(* CoDeSys 2.3.9.16 project: PLC_OPEN_test.pro *)
(* Libraries: SysLibTargetVisu.lib 22.7.09 19:44:32, ANALYZATION.LIB 22.7.09 19:44:32, SysLibSockets.lib 22.7.09 19:44:32, SysLibCom.lib 22.7.09 19:44:32, SysLibTime.lib 22.7.09 19:44:32, AD_Convertor.lib 8.4.16 09:37:26, CPAC_TCP.lib 26.6.14 15:50:29, Standard.lib 22.7.09 19:44:32, IecSfc.lib 22.7.09 19:44:32, CPAC GUC-X00-TPX.lib 28.10.10 10:45:18, SysLibMem.lib 22.7.09 19:44:32, SysTaskInfo.lib 22.7.09 19:44:32, SYSLIBCALLBACK.LIB 22.7.09 19:44:32, 3S_CANopenMaster.lib 28.10.13 11:32:40, 3S_CANopenManager.lib 28.10.13 11:32:40, 3S_CanDrv.lib 28.10.13 11:32:40 *)

(* Task configuration *)
TASK PLC_PRG_TASK (PRIORITY := 1, INTERVAL := T#30ms);
	PLC_PRG
	RT_Manager
	TiltManager
	LiftManager
END_TASK
TASK VISU_TASK (PRIORITY := 15, INTERVAL := T#800ms);
	MAINTARGETVISU_PAINT_CODE
END_TASK
TASK SensorRead (PRIORITY := 10, INTERVAL := T#30ms);
	SensorRead();
END_TASK
TASK VISU_INPUT_TASK (PRIORITY := 14, INTERVAL := T#50ms);
	MAINTARGETVISU_INPUT_CODE
END_TASK

(* Global variable list: CanOpen implicit Variables *)
VAR_GLOBAL CONSTANT
	MAX_CTRLINDEX : INT := 0;
END_VAR
VAR_GLOBAL CONSTANT
	USE_CANOPEN_NODES : BOOL := TRUE;
	MAX_MASTERINDEX : INT := 0;
	MAX_NODEINDEX : INT := 1;
	MAX_SDOINDEX : INT := 65;
	MAX_PDOINDEX_RX : INT := 7;
	MAX_PDOINDEX_TX : INT := 7;
	MAX_MASTER_ODENTRY_IDX : INT := 0;
END_VAR
VAR_GLOBAL
	pCANopenMaster : ARRAY[0..MAX_MASTERINDEX] OF CanOpenMaster;
	pCanOpenNode : ARRAY[0..MAX_NODEINDEX] OF CanOpenNode;
	pCanOpenSDO : ARRAY[0..MAX_SDOINDEX] OF CanOpenSDO;
	pCanOpenPDO_Rx : ARRAY[0..MAX_PDOINDEX_RX] OF CanOpenPDO_Rx;
	pCanOpenPDO_Tx : ARRAY[0..MAX_PDOINDEX_TX] OF CanOpenPDO_Tx;
	 ODMEntries: ARRAY[0..MAX_MASTER_ODENTRY_IDX] OF CanOpenODEntry;
END_VAR

(* Global variable list: CANopen_MC_GLB *)
VAR_GLOBAL
	g_CAN_udiStationAmount:UDINT;	(*driver amount on the bus*)
	g_CAN_arAxis: ARRAY [1..255] OF TAxisStatus;	(*0:no mode 1:PP mode 2:PV mode 3:TC mode 4:Homing*)
END_VAR

(* Global variable list: Global_Variables *)
VAR_GLOBAL
	ComHandle: DWORD;
	byRead:ARRAY[1..16]OF BYTE;
	diSocket: DINT:= SOCKET_INVALID;(*SOCKET_INVALID=-1,DINT类型,FFFFFFFF,*)
	xRelativeExe1,xRelativeExe2: BOOL;
	xPowerOn1,xPowerOn2: BOOL;
	xPowerOff1,xPowerOff2: BOOL;
	xStop1,xStop2: BOOL;
	xVelocityExe1,xVelocityExe2: BOOL;
	xReset1,xReset2: BOOL;
	diVelocity1: UDINT:=20000;
	diPosition1,diPosition2: DINT;
	diVelocity2: UDINT:= 20000;
	diVelocity_jog1,diVelocity_jog2: DINT;
	Acc,Dec:DINT;(*加/减速度*)
	ENC_POS1: LREAL;(*病床磁条编码器读数*)
	ENC_POS2: LREAL;(*旋转部编码器读数*)
	ENC_Value: DINT;(*检测到INDEX信号时外部编码器的读数*)
	Client0,Client1,Client2: CLIENT_ACCEPT;
	LiftSpeed:UINT;
	Input_Value:DINT;
	Move_Height:REAL;
	Move_Angle:REAL;

	gLastLiftAngle:REAL;
	gLiftMotionState:UINT:=0;
END_VAR

(* Data type *)
TYPE TAxisStatus :
STRUCT
	usiAxis:USINT;			(*Axis address*)
	usiCurrentMode:USINT;	(*current motion mode*)


END_STRUCT
END_TYPE

(* POU 主程序/PLC_PRG, ST *)
PROGRAM PLC_PRG
VAR
	uiPort: UINT:= 5000;
	bActive: BOOL:=TRUE;
	ON:BOOL:=TRUE;
	RO:ARRAY [1..5] OF BYTE:=16#52,16#4F,16#00,16#5C,16#2D;
	RC:ARRAY [1..7] OF BYTE:=16#52,16#43,16#01,16#00,16#FF,16#31,16#8D;
	ROON,RCON:UINT;
	ComUseTimer:TON;
	cs:COMSETTINGS;(*RS232通讯*)
	bInit,bExit,open,close: BOOL;
	ComFilter:ComFilter;

	byReadRO:ARRAY [1..16] OF BYTE;
	ENC_Status:INT;
	LastIndexVelue:DINT;
	Offset: ARRAY [1..10] OF DINT;
	i:DINT;
	asda: DINT;
END_VAR
IF ON THEN(*寄存器初始化*)
	RegisterCallbacks();
	bInit:=TRUE;
	ON:=FALSE;
END_IF
IF bInit  THEN(* Open COM interface *)
	bInit:=FALSE;bExit:=FALSE;
	cs.	Port:=COM2;
	cs.dwBaudRate:=38400;
	cs.byParity:=0;
	cs.byStopBits:=1;
	cs.dwBufferSize:=1024;
	ComHandle := SysComOpen(cs.Port);
	IF ComHandle<> INVALID_HANDLE THEN(* INVALID_HANDLED，常数，代表32位FFFFFFFF*)
		open := SysComSetSettings(ComHandle, ADR(cs));(*OPEN=1，串口处于正常打开状态*)
		IF open THEN
			close:=FALSE;
		END_IF
	ELSE
		bExit:=TRUE;
	END_IF
END_IF
IF bExit THEN(* Close COM interface *)
	bExit:=FALSE;bInit:=FALSE;
	close := SysComClose(ComHandle);(*close=1，串口处于关闭状态*)
	ComHandle:=0;
	IF close THEN
		open:=FALSE;
	END_IF
END_IF
ComFilter();
CASE ROON OF(*ROON：RO指令发送和接收具体步骤*)
0:	ComUseTimer(IN:=TRUE,PT:=t#3s);
	IF ComUseTimer.Q THEN
		ROON:=1;
		ComUseTimer(IN:=FALSE,PT:=t#3s);
	END_IF
1:	SysComWrite(ComHandle, ADR(RO), 5, 5);	(*发送RO指令*)
	ROON:=2;
2:	IF byRead[1]=16#52 AND byRead[2]=16#4F THEN
		byReadRO:=byRead;
		ROON:=3;
		ComUseTimer(IN:=FALSE,PT:=t#3s);
	END_IF
	ComUseTimer(IN:=TRUE,PT:=t#3s);
	IF ComUseTimer.Q THEN
		ROON:=99;
		ComUseTimer(IN:=FALSE,PT:=t#3s);
	END_IF
3:	IF   byReadRO[1]=16#52 AND byReadRO[2]=16#4F AND byReadRO[3]=16#06 THEN(*判断接收每个字节的内容，该语句判断为正确的回码*)
		ROON:=4;
		RCON:=1;			(*ROON为4证明RO指令发送成功,RCON=1，开始发送RC指令*)
	ELSIF byReadRO[1]=16#52 AND byReadRO[2]=16#4F AND byReadRO[3]<>16#06THEN(*判断接收前三个字节的内容，该语句判断为错误的回码*)
		ROON:=100;(*步骤停止在100并报错*)
	END_IF
END_CASE
CASE RCON OF
1:	SysComWrite(ComHandle, ADR(RC), 7, 5);(*发送RC指令*)
	RCON:=2;
2:	ComUseTimer(IN:=TRUE,PT:=t#250ms);(*定时器*)
	IF ComUseTimer.Q THEN(*定时250ms到，发送一次RC指令*)
		RCON:=1;
		ComUseTimer(IN:=FALSE,PT:=t#250ms);(*定时器*)
	END_IF
END_CASE
IF bActive THEN
	IF diSocket = SOCKET_INVALID THEN
		diSocket := TcpServerOpenSocket(uiPort, 3);(*TCP/IP设置，按F1可查看功能解释*)
	ELSE
		IF Client0.diSocket = SOCKET_INVALID THEN
			Client0:= TcpServerWaitForConnect(diSocket, 200);
		END_IF
		IF Client1.diSocket = SOCKET_INVALID THEN
			Client1:= TcpServerWaitForConnect(diSocket, 200);
		END_IF
		IF Client2.diSocket = SOCKET_INVALID THEN
			Client2:= TcpServerWaitForConnect(diSocket, 200);
		END_IF
	END_IF
ELSE
	IF diSocket <> SOCKET_INVALID THEN(*关闭服务器连接端口*)
		CloseSocket(ADR(diSocket));
		IF Client0.diSocket <> SOCKET_INVALID THEN
			CloseSocket(ADR(Client0.diSocket));
			Client0.stIPAddress:= '';
		END_IF
		IF Client1.diSocket <> SOCKET_INVALID THEN
			CloseSocket(ADR(Client1.diSocket));
			Client1.stIPAddress:= '';
		END_IF
		IF Client2.diSocket <> SOCKET_INVALID THEN
			CloseSocket(ADR(Client2.diSocket));
			Client2.stIPAddress:= '';
		END_IF
	END_IF
END_IF
GT_GetEncPos(9, ADR(ENC_POS1), 1, 0);	(*读取编码器位置：病床平移编码器*)
GT_GetEncPos(4, ADR(ENC_POS2), 1, 0);	(*读取编码器位置：机架旋转部编码器*)
GT_SetCaptureMode(4,CAPTURE_INDEX);	(*F1查询函数定义*)
GT_GetCaptureStatus(4, ADR(ENC_Status), ADR(ENC_Value), 1,0);(*读取编码器捕获状态：读取机架编码器Index信号*)
GT_GetDi(MC_GPI,ADR(Input_Value));(*读取端子板数字输入口信息*)
IF ENC_Value>0AND(ENC_Value/5760)<1 AND i<=10THEN
	LastIndexVelue:=ENC_Value;
ELSIF (ENC_Value/5760)>1 AND i<=10THEN
	IF ENC_Value<>LastIndexVelue  THEN
		IF ((ENC_Value-LastIndexVelue)<>5760)THEN
			i:=i+1;
			Offset[i]:=ENC_Value-LastIndexVelue;
			LastIndexVelue:=ENC_Value;
		ELSE
			LastIndexVelue:=ENC_Value;
		END_IF
	END_IF
END_IF
END_PROGRAM

(* POU PLCOpen_CAN2.3/串口通讯/ComFilter, ST *)
FUNCTION_BLOCK ComFilter
VAR_INPUT
END_VAR
VAR_OUTPUT
END_VAR
VAR
	NullArray,Buffer,MyBuffer:ARRAY [1..16] OF BYTE;
	ComRecieveBytes,MyRecieveBytes:DWORD;
	i:UINT:=0;
	j,k,l,m,n:UINT;
END_VAR
IF ComHandle<> INVALID_HANDLE THEN
	ComRecieveBytes:=SysComRead(ComHandle,ADR(Buffer) , 12, 1);(*串口接收*)
	IF i=1 THEN
		IF  ComRecieveBytes=4 THEN
			IF	Buffer[1]<>16#47 THEN
				MyBuffer[2]:=Buffer[1];
				MyBuffer[3]:=Buffer[2];
				MyBuffer[4]:=Buffer[3];
				MyBuffer[5]:=Buffer[4];
				byRead:=MyBuffer;
				MyBuffer:=NullArray;
				i:=0;

			(*ELSE
				MyBuffer:=NullArray;
				i:=0;*)
			END_IF
		ELSIF ComRecieveBytes>4  THEN
			IF	Buffer[1]=16#47 THEN
				MyBuffer[2]:=Buffer[1];
				MyBuffer[3]:=Buffer[2];
				MyBuffer[4]:=Buffer[3];
				MyBuffer[5]:=Buffer[4];
				MyBuffer[6]:=Buffer[5];
				MyBuffer[7]:=Buffer[6];
				MyBuffer[8]:=Buffer[7];
				MyBuffer[9]:=Buffer[8];
				byRead:=MyBuffer;
				MyBuffer:=NullArray;
				i:=0;
			(*ELSE
				MyBuffer:=NullArray;
				i:=0;*)
			END_IF
		END_IF
	ELSIF i=2 THEN
		IF  ComRecieveBytes=5-MyRecieveBytes THEN
			MyBuffer[MyRecieveBytes+1]:=Buffer[1];
			MyBuffer[MyRecieveBytes+2]:=Buffer[2];
			MyBuffer[MyRecieveBytes+3]:=Buffer[3];
			MyBuffer[MyRecieveBytes+4]:=Buffer[4];
			MyBuffer[MyRecieveBytes+5]:=Buffer[5];
			byRead:=MyBuffer;
			MyBuffer:=NullArray;
			MyRecieveBytes:=0;
			i:=0;
		(*ELSE
			MyBuffer:=NullArray;
			MyRecieveBytes:=0;
			i:=0;*)
		END_IF
	ELSIF i=3 THEN
		IF  ComRecieveBytes=9-MyRecieveBytes THEN
			MyBuffer[MyRecieveBytes+1]:=Buffer[1];
			MyBuffer[MyRecieveBytes+2]:=Buffer[2];
			MyBuffer[MyRecieveBytes+3]:=Buffer[3];
			MyBuffer[MyRecieveBytes+4]:=Buffer[4];
			MyBuffer[MyRecieveBytes+5]:=Buffer[5];
			MyBuffer[MyRecieveBytes+6]:=Buffer[6];
			MyBuffer[MyRecieveBytes+7]:=Buffer[7];
			byRead:=MyBuffer;
			MyBuffer:=NullArray;
			MyRecieveBytes:=0;
			i:=0;
		(*ELSE
			MyBuffer:=NullArray;
			MyRecieveBytes:=0;
			i:=0;*)
		END_IF
	END_IF
	IF i=0 AND ComRecieveBytes=1 AND Buffer[1]=16#52 THEN
		MyBuffer:=Buffer;
		Buffer:=NullArray;
		i:=1;
	ELSIF i=0 AND ComRecieveBytes>1AND ComRecieveBytes<5 AND Buffer[1]=16#52THEN
		IF  Buffer[2]<>16#47 THEN
			MyBuffer:=Buffer;
			MyRecieveBytes:=ComRecieveBytes;
			Buffer:=NullArray;
			i:=2;
		ELSIF	 Buffer[2]=16#47 THEN
			MyBuffer:=Buffer;
			MyRecieveBytes:=ComRecieveBytes;
			Buffer:=NullArray;
			i:=3;
		END_IF
	ELSIF	i=0 AND ComRecieveBytes=5 AND Buffer[1]=16#52 THEN
		IF Buffer[2]<>16#47 THEN
			byRead:=Buffer;
			Buffer:=NullArray;
		ELSIF  Buffer[2]=16#47 THEN
			MyBuffer:=Buffer;
			MyRecieveBytes:=ComRecieveBytes;
			Buffer:=NullArray;
			i:=3;
		END_IF
	ELSIF  i=0 AND ComRecieveBytes>5 AND ComRecieveBytes<9  AND Buffer[1]=16#52 AND  Buffer[2]=16#47THEN
		MyBuffer:=Buffer;
		MyRecieveBytes:=ComRecieveBytes;
		Buffer:=NullArray;
		i:=3;
	ELSIF i=0 AND ComRecieveBytes=9  AND Buffer[1]=16#52 AND  Buffer[2]=16#47THEN
			byRead:=Buffer;
			Buffer:=NullArray;
	END_IF
END_IF
END_FUNCTION_BLOCK

(* POU 子程序/RT_Manager, ST *)
PROGRAM RT_Manager
VAR
	fbRelMove1,fbRelMove2: MC_MoveRelative;
	fbPower1,fbPower2: MC_Power;
	fbStop1,fbStop2: MC_Stop;
	fbVelMove1,fbVelMove2:MC_MoveVelocity;
	fbReset1,fbReset2: MC_Reset;
	LanNullArray,abyRecvRaw,abyRecv,HeartBeat: ARRAY [1..256] OF BYTE;
	diReceived:DINT;
	diRotateHomestep,diRotateJogstep,diRotateMovetostep,diRotateStopstep:UINT;
	diTraverseHomestep,diTraverseJogstep,diTraverseMovetostep,diTraverseStopstep:UINT;
	SizeOfMsg:INT;
	RotateFirstPos,FirstIndexPos:DINT;
	TraverseFirstPos:DINT;
	TargetPosition:LREAL;
	str1: STRING(50):= 'HOME ROTATE;ACK@';str2: STRING(50):= 'HOME ROTATE;UNDERWAY@';str3: STRING(50):= 'HOME ROTATE;COMPLETED@';str4: STRING(50):= 'HOME ROTATE; FAILED=';
	str5: STRING(50):= 'JOG ROTATE;ACK@';str6: STRING(50):= 'JOG ROTATE;UNDERWAY@';str7: STRING(50):= 'JOG ROTATE;COMPLETED@';str8: STRING(50):= 'JOG ROTATE;FAILED=';
	str9: STRING(50):= 'MOVETO ROTATE;ACK@';str10: STRING(50):= 'MOVETO ROTATE;UNDERWAY@';str11: STRING(50):= 'MOVETO ROTATE;COMPLETED@';str12: STRING(50):= 'MOVETO ROTATE;FAILED=';
	str13: STRING(50):= 'STOP ROTATE;ACK@';str14: STRING(50):= 'STOP ROTATE;UNDERWAY@';str15: STRING(50):= 'STOP ROTATE;COMPLETED@';str16: STRING(50):= 'JOG ROTATE;STOPPED@';str17: STRING(50):= 'STOP ROTATE;FAILED=';
	str25: STRING(50):= 'RESET ROTATE;COMPLETED@';str26: STRING(50):= 'RESET ROTATE;FAILED=';
	str30: STRING(50):='HOME ROTATE;STOPPED@';str31: STRING(50):= 'MOVETO ROTATE;STOPPED@';str32: STRING(50):= 'GET ROTATE;COMPLETED;COUNTER =';

	str51: STRING(50):= 'HOME TRAVERSE;ACK@';str52: STRING(50):= 'HOME TRAVERSE;UNDERWAY@';str53: STRING(50):= 'HOME TRAVERSE;COMPLETED@';str54: STRING(50):= 'HOME TRAVERSE; FAILED=';
	str55: STRING(50):= 'JOG TRAVERSE;ACK@';str56: STRING(50):= 'JOG TRAVERSE;UNDERWAY@';str57: STRING(50):= 'JOG TRAVERSE;COMPLETED@';str58: STRING(50):= 'JOG TRAVERSE;FAILED=1@';
	str59: STRING(50):= 'MOVETO TRAVERSE;ACK@';str60: STRING(50):= 'MOVETO TRAVERSE;UNDERWAY@';str61: STRING(50):= 'MOVETO TRAVERSE;COMPLETED@';str62: STRING(50):= 'MOVETO TRAVERSE;FAILED=1@';
	str63: STRING(50):= 'STOP TRAVERSE;ACK@';str64: STRING(50):= 'STOP TRAVERSE;UNDERWAY@';str65: STRING(50):= 'STOP TRAVERSE;COMPLETED@';str66: STRING(50):= 'JOG TRAVERSE;STOPPED@';
	str67: STRING(50):= 'MOVETO TRAVERSE;STOPPED@';str68: STRING(50):= 'HOME TRAVERSE;STOPPED@'; str69: STRING(50):= 'STOP TRAVERSE;FAILED=';
	str73: STRING(50):= 'SET TRAVERSE;COMPLETED@';str74: STRING(50):= 'SET TRAVERSE;FAILED=';

	str77: STRING(50):= 'RESET TRAVERSE;COMPLETED@';str78: STRING(50):= 'RESET TRAVERSE;FAILED=';str79:STRING(50):='JOG TRAVERSE;FAILED=Forward sw Limit@';
	str80:STRING(50):='JOG TRAVERSE;FAILED=Reverse sw Limit@';
	i,j,k,SecondColonPos: INT;
	Temp,Temp1,Temp2,Temp3: STRING;
	RotatePosition,RotateSpeed,RotateTurns,TraversePosition,TraverseSpeed: STRING;
	Horz_Limit_Home,Horz_Limit_In,Horz_Limit_Out:UINT;
	RotateUseTimer1,RotateUseTimer2,RotateUseTimer3,TraverseUseTimer1,TraverseUseTimer2,TraverseUseTimer3:TON;(*信息处理超时*)
	MoveOverTime,AutoSendMsgDelay,HeartBeatTimer:TON;
	AutoSendMsgStep:UINT:=0;
	HeartBeatStep,HeartBeatCounts: INT;
	EmergencyStop: INT;
	OneAngleToPulse: LREAL:=323.9;
END_VAR
IF	 Client0.diSocket <> SOCKET_INVALID THEN
	diReceived:= TcpReceiveData(Client0.diSocket, ADR(abyRecvRaw), SIZEOF(abyRecvRaw), 10);
	IF diReceived>0 THEN
		IF abyRecvRaw[1]=16#52 AND abyRecvRaw[2]=16#54 AND diReceived=22THEN
			HeartBeat:=abyRecvRaw;
			abyRecvRaw:=LanNullArray;
		ELSIF (abyRecvRaw[1]<>16#52 OR abyRecvRaw[2]<>16#54) AND( abyRecvRaw[diReceived-5]<>16#42 OR abyRecvRaw[diReceived-4]<>16#45 OR abyRecvRaw[diReceived-3]<>16#41 OR abyRecvRaw[diReceived-2]<>16#54)THEN
			SizeOfMsg:=DINT_TO_INT(diReceived-2);
			abyRecv:=abyRecvRaw;
			abyRecvRaw:=LanNullArray;
		ELSIF abyRecvRaw[1]=16#52 AND abyRecvRaw[2]=16#54 AND diReceived<>22THEN
			FOR i:=1TO (DINT_TO_INT(diReceived)) BY 1 DO
				IF i<=20 THEN
					HeartBeat[i]:=abyRecvRaw[i];
				END_IF
				IF i>=23 THEN
					abyRecv[i-22]:=abyRecvRaw[i];
				END_IF
				IF  i=diReceived THEN
					abyRecvRaw:=LanNullArray;
				END_IF
			END_FOR
			SizeOfMsg:=DINT_TO_INT(diReceived-24);
		ELSIF abyRecvRaw[1]<>16#52 AND abyRecvRaw[2]<>16#54 AND abyRecvRaw[diReceived-5]=16#42 AND abyRecvRaw[diReceived-4]=16#45 AND abyRecvRaw[diReceived-3]=16#41 AND abyRecvRaw[diReceived-2]=16#54THEN
			FOR i:=1 TO (DINT_TO_INT(diReceived-24))  BY 1 DO
				abyRecv[i]:=abyRecvRaw[i];
			END_FOR
			FOR i:=1 TO 20 BY 1 DO
				HeartBeat[i]:=abyRecvRaw[diReceived-22+i];
			END_FOR
			SizeOfMsg:=DINT_TO_INT(diReceived-24);
			abyRecvRaw:=LanNullArray;
		END_IF
		(*Heart Beat*)
		IF HeartBeat[1]=16#52 AND HeartBeat[2]=16#54 AND HeartBeat[3]=16#4D AND HeartBeat[4]=16#61 AND HeartBeat[5]=16#6E AND HeartBeat[6]=16#61 AND  HeartBeat[7]=16#67 AND HeartBeat[8]=16#65 AND HeartBeat[9]=16#72 THEN
			HeartBeatStep:=1;
			HeartBeatCounts:=HeartBeatCounts+1;
		END_IF
	(*Rotate:版本信息*)
		IF abyRecv[1]=86 AND abyRecv[2]=69AND abyRecv[3]=82 AND abyRecv[4]=83AND abyRecv[5]=73AND abyRecv[6]=79AND abyRecv[7]=78AND abyRecv[8]=32AND abyRecv[9]=82AND abyRecv[10]=79AND abyRecv[11]=84AND abyRecv[12]=65AND abyRecv[13]=84AND abyRecv[14]=69THEN
			Temp:='';
			Temp:='VERSION ROTATE;<version STRING>@';
			TcpSendData(Client0.diSocket, ADR(Temp), LEN(Temp), 10);
			abyRecv:=LanNullArray;
		END_IF
	(*Traverse：获取版本信息*)
		IF((abyRecv[1]=86)AND(abyRecv[2]=69)AND(abyRecv[3]=82)AND(abyRecv[4]=83)AND(abyRecv[5]=73)AND(abyRecv[6]=79)AND(abyRecv[7]=78)AND(abyRecv[8]=32)AND(abyRecv[9]=84 ) AND(abyRecv[10]=82) AND(abyRecv[11]=65 ) AND(abyRecv[12]=86) AND(abyRecv[13]=69) AND(abyRecv[14]=82) AND(abyRecv[15]=83) AND(abyRecv[16]=69) )THEN
			Temp:='';
			Temp:='VERSION TRAVERSE;<version STRING>@';
			TcpSendData(Client0.diSocket, ADR(Temp), LEN(Temp), 0);
			abyRecv:=LanNullArray;
		END_IF
		IF diRotateStopstep=0 THEN
		(*Rotate:Stop动作*)
			IF abyRecv[1]=83AND abyRecv[2]=84AND abyRecv[3]=79 AND abyRecv[4]=80 AND abyRecv[5]=32AND abyRecv[6]=82 AND abyRecv[7]=79AND abyRecv[8]=84AND abyRecv[9]=65AND abyRecv[10]=84AND abyRecv[11]=69 THEN(*判断为Gantry stop命令*)
				TcpSendData(Client0.diSocket, ADR(str13), LEN(str13), 10);(*通过客户端0发送字符串13（STOP ROTATE;ACK）*)
				IF  diRotateJogstep>0 THEN(*如果JOG动作正在执行*)
					diRotateStopstep:=1;diRotateJogstep:=0;xVelocityExe1:=FALSE;
					TcpSendData(Client0.diSocket, ADR(str16), LEN(str16), 10);
				ELSIF  diRotateHomestep>0 THEN(*如果HOME动作正在执行*)
					diRotateStopstep:=20;diRotateHomestep:=0;
					TcpSendData(Client0.diSocket, ADR(str30), LEN(str30), 10);
				ELSIF diRotateMovetostep>0 THEN(*如果MOVETO动作正在执行*)
					diRotateStopstep:=30;diRotateMovetostep:=0;
					TcpSendData(Client0.diSocket, ADR(str31), LEN(str31), 10);
				ELSIF diRotateHomestep=0 AND diRotateMovetostep=0 AND diRotateJogstep=0 THEN(*如果没有任何动作正在执行*)
					diRotateStopstep:=40;
				END_IF
				abyRecv:=LanNullArray;
			ELSIF diRotateHomestep=0 AND diRotateMovetostep=0 AND (diRotateJogstep=0OR diRotateJogstep=4)THEN
			(*Rotate:Home动作*)
				IF abyRecv[1]=72 AND abyRecv[2]=79AND abyRecv[3]=77 AND abyRecv[4]=69 AND abyRecv[5]=32AND abyRecv[6]=82 AND abyRecv[7]=79AND abyRecv[8]=84AND abyRecv[9]=65AND abyRecv[10]=84AND abyRecv[11]=69THEN
					IF ENC_Value<ENC_POS2 OR (ENC_Value=0 AND ENC_POS2 =0)THEN(*满足任一条件：上电后机架已转动过，当前不在Index位置或者系统刚上电机架未转动过*)
						FirstIndexPos:=ENC_Value;(*记录当前滑环编码器index读数*)
						diVelocity_jog1:=-4000;Acc:=4000;Dec:=1000;
						xVelocityExe1:=TRUE;diRotateHomestep:=1;
					ELSIF ENC_Value=ENC_POS2 AND ENC_Value<>0 AND ENC_POS2 <>0THEN(*满足2个条件：1、当前处在在Index位置2、系统上电后机架已转动过 *)
						diRotateHomestep:=3;(*机架不需要旋转，直接回COMPLETE*)
					END_IF
					TcpSendData(Client0.diSocket, ADR(str1), LEN(str1), 10);
					TcpSendData(Client0.diSocket, ADR(str2), LEN(str2), 10);
					abyRecv:=LanNullArray;
			(*Rotate:Moveto动作*)
				ELSIF  abyRecv[1]=77 AND abyRecv[2]=79AND abyRecv[3]=86 AND abyRecv[4]=69AND abyRecv[5]=84AND abyRecv[6]=79AND abyRecv[7]=32AND abyRecv[8]=82AND abyRecv[9]=79AND abyRecv[10]=84AND abyRecv[11]=65AND abyRecv[12]=84 AND abyRecv[13]=69THEN
					Temp1:='';
					FOR j:=1 TO SizeOfMsg DO
						Temp1:=CONCAT(Temp1,ASCII_TO_STRING(abyRecv[j]));(*将命令内容转换为字符串存放在Temp1中*)
					END_FOR;
					TargetPosition:=STRING_TO_LREAL (DELETE(Temp1,24,1));(*目标位置*)
					IF	GR_POS(ENC_Value,ENC_POS2)>0 AND GR_POS(ENC_Value,ENC_POS2)<888.8 THEN
						IF (TargetPosition-GR_POS(ENC_Value,ENC_POS2))>5.0 AND (TargetPosition<>0) THEN(*如果满足2个条件：1、目标位置大于当前位置且大于5°2、目标位置不是0°*)
							diPosition1:=LREAL_TO_DINT((TargetPosition-GR_POS(ENC_Value,ENC_POS2))*(-1*OneAngleToPulse));(*将机架的目标位置转换为电机的目标位置（脉冲数）；-323.9：负号表示电机逆时针转动机架顺时针转动，323.9表示机架旋转1°对应电机转动的脉冲数*)
							diVelocity1:=8000;Acc:=1200;Dec:=900;(*设置位置模式参数：电机速度=40rpm，加速度=6rpm/s，减速度=4.5rpm/s*)
							xRelativeExe1:=TRUE;(*执行功能块fbRelMove1，开始位置模式的运动*)
							RotateFirstPos:=diActPosition1;(*记录电机当前位置*)
							TcpSendData(Client0.diSocket, ADR(str9), LEN(str9), 10);
							TcpSendData(Client0.diSocket, ADR(str10), LEN(str10), 10);
							diRotateMovetostep:=1;
						ELSIF (TargetPosition-GR_POS(ENC_Value,ENC_POS2))<5.0 AND (TargetPosition<>0) THEN(*如果满足2个条件：1、目标位置大于当前位置且小于5°2、目标位置不是0°*)
							diPosition1:=LREAL_TO_DINT((360+TargetPosition-GR_POS(ENC_Value,ENC_POS2))*(-1*OneAngleToPulse));(*将机架的目标位置转换为电机的目标位置（脉冲数），机架会多转1圈*)
							diVelocity1:=8000;Acc:=1200;Dec:=900;
							xRelativeExe1:=TRUE;
							RotateFirstPos:=diActPosition1;
							TcpSendData(Client0.diSocket, ADR(str9), LEN(str9), 10);
							TcpSendData(Client0.diSocket, ADR(str10), LEN(str10), 10);
							diRotateMovetostep:=1;
						ELSIF (TargetPosition < GR_POS(ENC_Value,ENC_POS2))AND(TargetPosition<>0) THEN(*如果满足2个条件：1、目标位置小于当前位置且小于5°2、目标位置不是0°*)
							diPosition1:=LREAL_TO_DINT((360.0+TargetPosition-GR_POS(ENC_Value,ENC_POS2))*(-1*OneAngleToPulse));
							diVelocity1:=8000;Acc:=1200;Dec:=900;
							xRelativeExe1:=TRUE;
							RotateFirstPos:=diActPosition1;
							TcpSendData(Client0.diSocket, ADR(str9), LEN(str9), 10);
							TcpSendData(Client0.diSocket, ADR(str10), LEN(str10), 10);
							diRotateMovetostep:=1;
						ELSIF TargetPosition=0AND(360.0-GR_POS(ENC_Value,ENC_POS2))>5 THEN(*如果满足2个条件：1、当前位置距0°位置大于5° 2、目标位置是0°*)
							diPosition1:=LREAL_TO_DINT((360.0-GR_POS(ENC_Value,ENC_POS2))*(-1*OneAngleToPulse));
							diVelocity1:=8000;Acc:=1200;Dec:=900;
							xRelativeExe1:=TRUE;
							RotateFirstPos:=diActPosition1;
							TcpSendData(Client0.diSocket, ADR(str9), LEN(str9), 10);
							TcpSendData(Client0.diSocket, ADR(str10), LEN(str10), 10);
							diRotateMovetostep:=1;
						ELSIF TargetPosition=0AND(360.0-GR_POS(ENC_Value,ENC_POS2))<5 THEN(*如果满足2个条件：1、当前位置距0°位置小于5° 2、目标位置是0°*)
							diPosition1:=LREAL_TO_DINT((720.0-GR_POS(ENC_Value,ENC_POS2))*(-1*OneAngleToPulse));(*机架多走一圈*)
							diVelocity1:=8000;Acc:=1200;Dec:=900;
							xRelativeExe1:=TRUE;
							RotateFirstPos:=diActPosition1;
							TcpSendData(Client0.diSocket, ADR(str9), LEN(str9), 10);
							TcpSendData(Client0.diSocket, ADR(str10), LEN(str10), 10);
							diRotateMovetostep:=1;
						END_IF
					END_IF
					abyRecv:=LanNullArray;
			(*Rotate:Jog动作*)
				ELSIF abyRecv[1]=74AND abyRecv[2]=79 AND abyRecv[3]=71 AND abyRecv[4]=32 AND abyRecv[5]=82AND abyRecv[6]=79AND abyRecv[7]=84AND abyRecv[8]=65AND abyRecv[9]=84AND abyRecv[10]=69THEN
					Temp1:='';
					FOR j:=1 TO SizeOfMsg DO
						Temp1:=CONCAT(Temp1,ASCII_TO_STRING(abyRecv[j]));
					END_FOR
					diVelocity_jog1:=REAL_TO_DINT(STRING_TO_REAL (DELETE(Temp1,18,1)))*(-2000);(*将机架的目标速度转换为电机的目标速度（脉冲/ms)；-2000：负号表示电机逆时针转动机架顺时针转动，2000表示机架旋转1RPM对应电机转动100RPM=2000脉冲/ms*)
					Acc:=400000;Dec:=40000;(*加速度=2000rpm/s；减速度=200rpm/s*)
					TcpSendData(Client0.diSocket, ADR(str5), LEN(str5), 10);
					TcpSendData(Client0.diSocket, ADR(str6), LEN(str6), 10);
					diRotateJogstep:=1;
					abyRecv:=LanNullArray;
				END_IF
			END_IF
		END_IF
		(*Traverse:Stop动作*)
		IF abyRecv[1]=83 AND abyRecv[2]=84AND abyRecv[3]=79 AND abyRecv[4]=80 AND abyRecv[5]=32AND abyRecv[6]=84 AND abyRecv[7]=82AND abyRecv[8]=65AND abyRecv[9]=86AND abyRecv[10]=69AND abyRecv[11]=82AND abyRecv[12]=83AND abyRecv[13]=69THEN
			Temp3:='';
			FOR j:=1 TO SizeOfMsg DO
				Temp3:=CONCAT(Temp3,ASCII_TO_STRING(abyRecv[j]));
			END_FOR
			TcpSendData(Client0.diSocket, ADR(str63), LEN(str63), 10);
			xRelativeExe2:=FALSE;
			xVelocityExe2:=FALSE;
			xReset2:=FALSE;
			RotateUseTimer2(IN:=FALSE);
			IF diTraverseHomestep>0 THEN(*HOME动作正在执行中*)
				diTraverseHomestep:=0;
				TcpSendData(Client0.diSocket, ADR(str68), LEN(str68), 10);
			ELSIF diTraverseMovetostep>0 THEN(*MOVETO动作正在执行中*)
				diTraverseMovetostep:=0;
				TcpSendData(Client0.diSocket, ADR(str67), LEN(str67), 10);
			ELSIF diTraverseJogstep>0 THEN(*JOG动作正在执行中*)
				diTraverseJogstep:=0;
				TcpSendData(Client0.diSocket, ADR(str66), LEN(str66), 10);
			END_IF
			xStop2:=TRUE;
			diTraverseStopstep:=1;
			abyRecv:=LanNullArray;
		ELSIF(diTraverseHomestep+diTraverseJogstep+diTraverseMovetostep+diTraverseStopstep)=0 THEN
			 IF abyRecv[1]=72 AND abyRecv[2]=79AND abyRecv[3]=77 AND abyRecv[4]=69AND abyRecv[5]=32AND abyRecv[6]=84 AND abyRecv[7]=82AND abyRecv[8]=65AND abyRecv[9]=86AND abyRecv[10]=69AND abyRecv[11]=82AND abyRecv[12]=83AND abyRecv[13]=69THEN
				TcpSendData(Client0.diSocket, ADR(str51), LEN(str51), 10);
				TcpSendData(Client0.diSocket, ADR(str52), LEN(str52), 10);
				Horz_Limit_Home:=1-(DINT_TO_WORD(Input_Value) AND 256)/256;	(*水平：Home位置光电开关*)
				IF Horz_Limit_Home=1 THEN(*当前已经过了HOME位置*)
					diVelocity_jog2:=0;
				ELSIF Horz_Limit_Home=0 THEN(*当前未过了HOME位置*)
					diVelocity_jog2:=-268800;(*电机速度=1344RPM，逆时针旋转*)
				END_IF
				xVelocityExe2:=TRUE;
				diTraverseHomestep:=1;
				abyRecv:=LanNullArray;
			(*Traverse:Moveto动作*)
			ELSIF abyRecv[1]=77 AND abyRecv[2]=79AND abyRecv[3]=86 AND abyRecv[4]=69AND abyRecv[5]=84AND abyRecv[6]=79AND abyRecv[7]=32AND abyRecv[8]=84AND abyRecv[9]=82AND abyRecv[10]=65AND abyRecv[11]=86AND abyRecv[12]=69AND abyRecv[13]=82AND abyRecv[14]=83AND abyRecv[15]=69THEN
				Temp2:='';
				FOR j:=1 TO SizeOfMsg DO
				Temp2:=CONCAT(Temp2,ASCII_TO_STRING(abyRecv[j]));
				END_FOR
				FOR k:=1 TO SizeOfMsg DO(*判断第二个；的位置*)
					IF abyRecv[k]=16#3B THEN
						SecondColonPos:=k;
					END_IF
				END_FOR
				TcpSendData(Client0.diSocket, ADR(str59), LEN(str59), 10);
				TcpSendData(Client0.diSocket, ADR(str60), LEN(str60), 10);
				diPosition2:=LREAL_TO_DINT(ENC_POS1/100-STRING_TO_LREAL (DELETE(Temp2,SecondColonPos+9,1)))*3360;(*diPosition2>0，往里进;diPosition2<0，往外出;*)(*3360：病床水平移动1mm对应电机走过的3360个脉冲*)
				diVelocity2:=REAL_TO_DINT(STRING_TO_REAL (DELETE(DELETE(Temp2,SizeOfMsg,SecondColonPos),23,1))*3360);(*3360：病床水平移动1mm/s对应电机转速3360脉冲/ms*)
				xRelativeExe2:=TRUE;diTraverseMovetostep:=1;
				TraverseFirstPos:=diActPosition2;(*记录电机当前位置，单位为脉冲*)
				abyRecv:=LanNullArray;
			(*Traverse:Jog动作*)
			ELSIF abyRecv[1]=74 AND abyRecv[2]=79AND abyRecv[3]=71 AND abyRecv[4]=32AND abyRecv[5]=84AND abyRecv[6]=82AND abyRecv[7]=65AND abyRecv[8]=86AND abyRecv[9]=69AND abyRecv[10]=82AND abyRecv[11]=83AND abyRecv[12]=69THEN
				Temp2:='';
				TcpSendData(Client0.diSocket, ADR(str55), LEN(str55), 10);
				TcpSendData(Client0.diSocket, ADR(str56), LEN(str56), 10);
				FOR j:=1 TO SizeOfMsg DO
					Temp2:=CONCAT(Temp2,ASCII_TO_STRING(abyRecv[j]));
				END_FOR
				IF STRING_TO_UINT(DELETE(Temp2, SizeOfMsg-1, 1)) =1 THEN(*如果给定运动方向为1，代表病床向机架里面进*)
					diVelocity_jog2:=REAL_TO_DINT(STRING_TO_REAL (DELETE(DELETE(Temp2, SizeOfMsg, SizeOfMsg-7),20,1))*3360);(*符号为正*)
				ELSE
					diVelocity_jog2:=REAL_TO_DINT(STRING_TO_REAL (DELETE(DELETE(Temp2, SizeOfMsg, SizeOfMsg-7),20,1))*(-3360));(*符号为负*)
				END_IF
				xVelocityExe2:=TRUE;
				diTraverseJogstep:=1;
				abyRecv:=LanNullArray;
			END_IF
		END_IF
	ELSIF diReceived<0 THEN
		CloseSocket(ADR(Client0.diSocket));
		Client0.stIPAddress:= '';
		HeartBeatTimer(IN:=FALSE);
		AutoSendMsgDelay(IN:=FALSE,PT:=t#500ms);
	END_IF
	IF AutoSendMsgStep=0 THEN
		AutoSendMsgDelay(IN:=TRUE,PT:=t#500ms);
		IF AutoSendMsgDelay.Q THEN
			AutoSendMsgStep:=1;
			AutoSendMsgDelay(IN:=FALSE,PT:=t#500ms);
		END_IF
	END_IF
	IF AutoSendMsgStep=1 THEN
		RotatePosition:=CONCAT(CONCAT('GET ROTATE;COMPLETED; POSITION=',LREAL_TO_STRING(LREAL_TO_LREALDOTN(GR_POS(ENC_Value,ENC_POS2),3))),'@');
		IF	(diRotateHomestep+diRotateJogstep+diRotateMovetostep+diRotateStopstep)=0 THEN
			RotateSpeed:=CONCAT(CONCAT('GET ROTATE;COMPLETED; SPEED=','0'),'@');
		ELSE
			RotateSpeed:=CONCAT(CONCAT('GET ROTATE;COMPLETED; SPEED=',LREAL_TO_STRING(LREAL_TO_LREALDOTN(DINT_TO_LREAL(diActVelocity1)/(-2000.00),3))),'@');
		END_IF
		RotateTurns:=CONCAT(CONCAT('GET ROTATE;COMPLETED;COUNTER =',DINT_TO_STRING(ENC_Value/11520)),'@');
		TraversePosition:=CONCAT(CONCAT('GET TRAVERSE;COMPLETED; POSITION=',REAL_TO_STRING(LREAL_TO_LREALDOTN(ENC_POS1/100,3))),'@');
		IF (diTraverseHomestep+diTraverseJogstep+diRotateMovetostep+diTraverseStopstep)=0 THEN
			TraverseSpeed:=CONCAT(CONCAT( 'GET TRAVERSE;COMPLETED; SPEED=','0'),'@');
		ELSE
			TraverseSpeed:=CONCAT(CONCAT('GET TRAVERSE;COMPLETED; SPEED=',LREAL_TO_STRING(LREAL_TO_LREALDOTN((DINT_TO_LREAL(ABS(diActVelocity2)))/3360.00,3))),'@');
		END_IF
		TcpSendData(Client0.diSocket, ADR(RotatePosition), LEN(RotatePosition), 0);
		TcpSendData(Client0.diSocket, ADR(RotateSpeed), LEN(RotateSpeed), 0);
		TcpSendData(Client0.diSocket, ADR(RotateTurns), LEN(RotateTurns), 0);
		TcpSendData(Client0.diSocket, ADR(TraversePosition), LEN(TraversePosition), 0);
		TcpSendData(Client0.diSocket, ADR(TraverseSpeed), LEN(TraverseSpeed), 0);
		AutoSendMsgStep:=0;
	END_IF
END_IF
(*Rotate:Home动作执行*)
CASE diRotateHomestep OF
1:	IF ENC_Value>FirstIndexPos THEN(*当机架连续转动过程中Index值发生改变时*)
		 xStop1:=TRUE;(*机架停止转动*)
		diRotateHomestep:=2;
	END_IF
2:	IF ABS(diActVelocity1)<200THEN(*电机速度小于1rpm*)
		diRotateHomestep:=3;
	END_IF
3:	RotateUseTimer1(IN:=TRUE, PT:=T#200ms);
	IF RotateUseTimer1.Q THEN(*延时*)
		TcpSendData(Client0.diSocket, ADR(str3), LEN(str3), 10);(*发送complete回码*)
		diRotateHomestep:=0;
		xPowerOff1:=TRUE;
		RotateUseTimer1(IN:=FALSE);
	END_IF
END_CASE
(*Rotate:Moveto动作执行*)
CASE diRotateMovetostep OF
1:	IF (ABS (ABS(diPosition1)-ABS(RotateFirstPos-diActPosition1)) <10)  THEN(*电机走完设定位置*)
		diRotateMovetostep:=2;
	END_IF
2:	RotateUseTimer1(IN:= TRUE, PT:=T#200ms);
	IF RotateUseTimer1.Q THEN(*延时*)
		TcpSendData(Client0.diSocket, ADR(str11), LEN(str11), 10);(*发送complete回码*)
		diRotateMovetostep:=0;
		xPowerOff1:=TRUE;
		RotateUseTimer1(IN:=FALSE);
	END_IF
END_CASE
(*Rotate:Jog动作执行*)
CASE diRotateJogstep OF
1:	xVelocityExe1:=TRUE;
	diRotateJogstep:=2;
2:	IF ABS( diActVelocity1 - diVelocity_jog1)<200  THEN(*达到目标速度时*)
		diRotateJogstep:=3;
	END_IF
3:	RotateUseTimer1(IN:=TRUE , PT:=T#200ms);(*定时器*)
	IF RotateUseTimer1.Q THEN
		TcpSendData(Client0.diSocket, ADR(str7), LEN(str7), 10);(*发送complete回码*)
		diRotateJogstep:=4;
		RotateUseTimer1(IN:=FALSE);
	 END_IF
END_CASE
(*Rotate:Stop动作执行*)
CASE diRotateStopstep OF(*停止JOG动作*)
1:																							(*第1段减速*)
	IF ABS(diActVelocity1) >=200000AND ABS(diActVelocity1) <402000 THEN											(*1000rpm<=电机速度<2010rpm*)
		diVelocity_jog1:=0; Dec:=26000;xVelocityExe1:=TRUE;diRotateStopstep:=2;	(*Dec=130rpm/s*)
	ELSIF ABS(diActVelocity1) >=100000AND ABS(diActVelocity1) <200000 THEN										(*500rpm<=电机速度<1000rpm*)
		diVelocity_jog1:=0; Dec:=18000;xVelocityExe1:=TRUE;diRotateStopstep:=3;	(*Dec=90rpm/s*)
	ELSIF ABS(diActVelocity1) >=40000AND ABS(diActVelocity1) <100000 THEN										(*200rpm<=电机速度<500rpm*)
		diVelocity_jog1:=0; Dec:=12000;  xVelocityExe1:=TRUE;diRotateStopstep:=4;	(*Dec=60rpm/s*)
	ELSIF ABS(diActVelocity1) >=20000AND ABS(diActVelocity1) <40000 THEN											(*100rpm<=电机速度<200rpm*)
		diVelocity_jog1:=0; Dec:=8000;  xVelocityExe1:=TRUE;diRotateStopstep:=5;	(*Dec=40rpm/s*)
	ELSIF ABS(diActVelocity1) >=10000AND ABS(diActVelocity1) <20000 THEN											(*50rpm<=电机速度<100rpm*)
		diVelocity_jog1:=0; Dec:=5000;  xVelocityExe1:=TRUE;diRotateStopstep:=6;	(*Dec=25rpm/s*)
	ELSIF ABS(diActVelocity1)>=6000AND ABS(diActVelocity1) <10000 THEN											(*30rpm<=电机速度<50rpm*)
		diVelocity_jog1:=0; Dec:=3000;  xVelocityExe1:=TRUE;diRotateStopstep:=7;	(*Dec=15rpm/s*)
	ELSIF ABS(diActVelocity1) >=4000AND ABS(diActVelocity1) <6000 THEN											(*20rpm<=电机速度<30rpm*)
		diVelocity_jog1:=0; Dec:=2000;  xVelocityExe1:=TRUE;diRotateStopstep:=8;	(*Dec=10rpm/s*)
	ELSIF ABS(diActVelocity1) >=2000AND ABS(diActVelocity1) <4000 THEN											(*10rpm<=电机速度<20rpm*)
		diVelocity_jog1:=0; Dec:=1400;  xVelocityExe1:=TRUE;diRotateStopstep:=9;	(*Dec=7rpm/s*)
	ELSIF ABS(diActVelocity1) <2000 THEN																	(*电机速度<10rpm*)
		diVelocity_jog1:=0; Dec:=1000;    xVelocityExe1:=TRUE;diRotateStopstep:=10;	(*Dec=5rpm/s*)
	END_IF
2:	IF ABS(diActVelocity1)>=100000 AND ABS(diActVelocity1) <200000 THEN			(*第2段减速*)
		diVelocity_jog1:=0; Dec:=18000;xVelocityExe1:=TRUE;diRotateStopstep:=3;
		END_IF
3:	IF ABS(diActVelocity1) >=40000AND ABS(diActVelocity1) <100000 THEN				(*第3段减速*)
		diVelocity_jog1:=0; Dec:=12000;  xVelocityExe1:=TRUE;diRotateStopstep:=4;
	END_IF
4:	IF ABS(diActVelocity1) >=20000AND ABS(diActVelocity1) <40000 THEN				(*第4段减速*)
		diVelocity_jog1:=0; Dec:=8000;  xVelocityExe1:=TRUE;diRotateStopstep:=5;
	  END_IF
5:	IF ABS(diActVelocity1) >=10000AND ABS(diActVelocity1)<20000 THEN				(*第5段减速*)
		diVelocity_jog1:=0; Dec:=5000;  xVelocityExe1:=TRUE;diRotateStopstep:=6;
	 END_IF
6:	IF ABS(diActVelocity1) >=6000AND ABS(diActVelocity1) <10000 THEN				(*第6段减速*)
		diVelocity_jog1:=0; Dec:=3000;  xVelocityExe1:=TRUE;diRotateStopstep:=7;
	END_IF
7:	IF ABS(diActVelocity1) >=4000AND ABS(diActVelocity1) <6000 THEN					(*第7段减速*)
		diVelocity_jog1:=0; Dec:=2000;  xVelocityExe1:=TRUE;diRotateStopstep:=8;
	END_IF
8:	IF ABS(diActVelocity1) >=2000AND ABS(diActVelocity1) <4000 THEN					(*第8段减速*)
		diVelocity_jog1:=0; Dec:=1400;  xVelocityExe1:=TRUE;diRotateStopstep:=9;
	END_IF
9:	IF ABS(diActVelocity1) >=1000 AND ABS(diActVelocity1 )<2000THEN					(*第9段减速*)
		diVelocity_jog1:=0; Dec:=1000;    xVelocityExe1:=TRUE;diRotateStopstep:=10;
	END_IF
10:	IF ABS(diActVelocity1) <400 THEN													(*第10段减速*)
		diVelocity_jog1:=0; Dec:=0;    xVelocityExe1:=TRUE;diRotateStopstep:=100;
		TcpSendData(Client0.diSocket, ADR(str14), SIZEOF(str14), 10);(*发送stop underway*)
	END_IF
20,30,40:
	RotateUseTimer1(IN:=TRUE,PT:=t#200ms);(*停止moveto和home动作*)
	IF RotateUseTimer1.Q THEN
		TcpSendData(Client0.diSocket, ADR(str14), LEN(str14), 10);(*发送stop underway*)
		xStop1:=TRUE;
		diRotateStopstep:=100;
		RotateUseTimer1(IN:=FALSE);
	END_IF
100:
	IF (ABS(diActVelocity1))<=200 THEN
		RotateUseTimer1(IN:=TRUE, PT:=T#300ms);
		IF RotateUseTimer1.Q THEN
			TcpSendData(Client0.diSocket, ADR(str15), LEN(str15), 10);(*发送stop complete*)
			diRotateStopstep:=0;
			xPowerOff1:=TRUE;
			RotateUseTimer1(IN:=FALSE);
		END_IF
	END_IF
END_CASE
(*Traverse:Home动作执行*)
CASE diTraverseHomestep OF
1:	Horz_Limit_Home:=1-(DINT_TO_WORD(Input_Value) AND 256)/256;	(*水平：Home位置光电开关*)
	IF  Horz_Limit_Home=1  THEN
		diVelocity_jog2:=80000;
		xVelocityExe2:=TRUE;
		diTraverseHomestep:=2;
	END_IF
2:	Horz_Limit_Home:=1-(DINT_TO_WORD(Input_Value) AND 256)/256;	(*水平：Home位置光电开关*)
	IF  Horz_Limit_Home=0 THEN
		xVelocityExe2:=FALSE;
		xStop2:=TRUE;
		diTraverseHomestep:=3;
	END_IF
3:	 IF  ABS( diActVelocity2)<200 THEN
		diTraverseHomestep:=4;
	END_IF
4:	TraverseUseTimer1(IN:=TRUE, PT:=T#300ms);
	IF TraverseUseTimer1.Q THEN
		TcpSendData(Client0.diSocket, ADR(str53), LEN(str53), 10);
		GT_SetEncPos(9, 0);
		diTraverseHomestep:=0;
		TraverseUseTimer1(IN:=FALSE);
	END_IF
END_CASE
(*Traverse:Moveto动作执行*)
CASE diTraverseMovetostep OF
1:	IF (ABS (ABS(diActPosition2-TraverseFirstPos)-ABS(diPosition2)))<50 THEN(*准确到达目标位置，由速度模式切换到位置模式执行MOVETO时，位置误差有35个脉冲，始终以位置模式执行MOVETO,误差为0脉冲*)
		diTraverseMovetostep:=2;
	END_IF
2..4:
	TraverseUseTimer1(IN:=TRUE, PT:=T#300ms);
	IF TraverseUseTimer1.Q THEN
		IF diTraverseMovetostep=2 THEN
			TcpSendData(Client0.diSocket, ADR(str61), LEN(str61), 10);
		ELSIF diTraverseMovetostep=3 THEN
			TcpSendData(Client0.diSocket, ADR(str62), LEN(str62), 10);
		ELSIF diTraverseMovetostep=4 THEN
			TcpSendData(Client0.diSocket, ADR(str62), LEN(str62), 10);
		END_IF
		diTraverseMovetostep:=0;
		TraverseUseTimer1(IN:=FALSE);
	END_IF
END_CASE
(*Traverse:Jog动作执行*)
CASE diTraverseJogstep OF
1:	IF  ABS(diActVelocity2-diVelocity_jog2)<400 THEN
		diTraverseJogstep :=2;
	ELSIF ABS(diActVelocity2)>980000  THEN(*超速、飞车*)
		diTraverseJogstep :=3;
	END_IF
2..3:
	TraverseUseTimer1(IN:= TRUE, PT:=T#300ms);
	IF TraverseUseTimer1.Q THEN
		IF diTraverseJogstep=2 THEN
			TcpSendData(Client0.diSocket, ADR(str57), LEN(str57), 10);
		ELSIF diTraverseJogstep=3 THEN
			TcpSendData(Client0.diSocket, ADR(str58), LEN(str58), 10);
		END_IF
			diTraverseJogstep :=4;
		TraverseUseTimer1(IN:= FALSE);
	END_IF
5:	Horz_Limit_In:=1-(DINT_TO_WORD(Input_Value) AND 512)/512;		(*水平：负方向限位开关*)
	IF Horz_Limit_In=0 THEN(*限位开关为0时，停止运动*)
		TcpSendData(Client0.diSocket, ADR(str80), LEN(str80), 10);
		xStop2:=TRUE;
		diTraverseJogstep:=7;
	END_IF
6:	Horz_Limit_Out:=1-(DINT_TO_WORD(Input_Value) AND 1024)/1024;	(*水平：正方向限位开关*)
	IF Horz_Limit_Out=0 THEN(*限位开关为0时，停止运动*)
		TcpSendData(Client0.diSocket, ADR(str79), LEN(str79), 10);
		 xStop2:=TRUE;
		diTraverseJogstep:=7;
	END_IF
7:	TraverseUseTimer2(IN:=TRUE,PT:=t#10ms);
		IF TraverseUseTimer2.Q THEN
			xStop2:=FALSE;
			TraverseUseTimer2(IN:=FALSE,PT:=t#10ms);
			diTraverseJogstep:=0;
		END_IF
END_CASE
IF diTraverseJogstep>0AND diTraverseJogstep<5  THEN(*JOG动作过程中判断限位开关为1，反向运动直到限位开关为0*)
	Horz_Limit_In:=1-(DINT_TO_WORD(Input_Value) AND 512)/512;		(*水平：负方向限位开关*)
	Horz_Limit_Out:=1-(DINT_TO_WORD(Input_Value) AND 1024)/1024;	(*水平：正方向限位开关*)
	IF Horz_Limit_In=1 THEN
		diVelocity_jog2:=-80000;
		xVelocityExe2:=TRUE;
		diTraverseJogstep :=5;
	ELSIF   Horz_Limit_Out=1 THEN(*JOG动作过程中判断限位开关为1，反向运动直到限位开关为0*)
		diVelocity_jog2:=80000;
		xVelocityExe2:=TRUE;
		diTraverseJogstep :=6;
	END_IF
END_IF
(*Traverse:Stop动作执行*)
CASE diTraverseStopstep OF
1:	TraverseUseTimer1(IN:= TRUE, PT:=t#100ms);
	IF TraverseUseTimer1.Q THEN
		TcpSendData(Client0.diSocket, ADR(str64), LEN(str64), 10);
		diTraverseStopstep:=2;
		TraverseUseTimer1(IN:= FALSE);
	END_IF
2:	MoveOverTime(IN:=TRUE,PT:=t#500ms);
	IF	MoveOverTime.Q THEN
		xStop2:=TRUE;
		diTraverseStopstep:=3;
		MoveOverTime(IN:=FALSE);
	END_IF
	IF (ABS(diActVelocity2))<300AND  control2.8THEN
		diTraverseStopstep:=3;
		MoveOverTime(IN:=FALSE);
	END_IF
3:	TraverseUseTimer1(IN:= TRUE, PT:=t#200ms);
	IF TraverseUseTimer1.Q THEN
		xReset2:=TRUE;
		TcpSendData(Client0.diSocket, ADR(str65), LEN(str65), 10);
		TraverseUseTimer1(IN:= FALSE);
		diTraverseStopstep:=0;
	END_IF
END_CASE
IF	xVelocityExe1 THEN
	RotateUseTimer2(IN:=TRUE ,PT:=T#15ms);
	IF RotateUseTimer2.Q AND ((diRotateJogstep>0AND diRotateJogstep<4)OR (diRotateHomestep>0)OR (diRotateStopstep>0)) THEN
		xVelocityExe1:=FALSE;
		RotateUseTimer2(IN:=FALSE);
	END_IF
END_IF
IF	xRelativeExe1 THEN
	RotateUseTimer2(IN:=TRUE ,PT:=T#15ms);
	IF RotateUseTimer2.Q AND diRotateMovetostep>0 THEN
		xRelativeExe1:=FALSE;
		RotateUseTimer2(IN:=FALSE);
	END_IF
END_IF
IF xStop1 THEN
	RotateUseTimer2(IN:=TRUE ,PT:=T#15ms);
	IF RotateUseTimer2.Q AND (diRotateHomestep>0 OR diRotateStopstep>0)  THEN
		xStop1:=FALSE;
		RotateUseTimer2(IN:=FALSE);
	END_IF
END_IF
RotateUseTimer3(IN:=xPowerOff1,PT:=T#15ms);
IF RotateUseTimer3.Q THEN
	xPowerOff1:=FALSE;
END_IF
IF	xVelocityExe2 THEN
	TraverseUseTimer2(IN:=TRUE,PT:=t#10ms);
	IF	TraverseUseTimer2.Q AND(diTraverseHomestep>0 OR diTraverseJogstep>0) THEN
		xVelocityExe2:=FALSE;
		TraverseUseTimer2(IN:=FALSE);
	END_IF
END_IF
IF	xRelativeExe2 THEN
	TraverseUseTimer2(IN:=TRUE,PT:=t#10ms);
	IF	TraverseUseTimer2.Q AND diTraverseMovetostep>0 THEN
		xRelativeExe2:=FALSE;
		TraverseUseTimer2(IN:=FALSE);
	END_IF
END_IF
IF	xStop2 THEN
	TraverseUseTimer3(IN:=TRUE,PT:=t#10ms);
	IF	TraverseUseTimer3.Q THEN
		xStop2:=FALSE;
		TraverseUseTimer3(IN:=FALSE);
	END_IF
END_IF
IF HeartBeatCounts>0 THEN
	HeartBeatTimer(IN:=TRUE,PT:=t#2s);
	IF HeartBeatStep=1 THEN
		HeartBeat:=LanNullArray;
		HeartBeatTimer(IN:=FALSE);
		EmergencyStop:=0;
		HeartBeatStep:=0;
	END_IF
	IF HeartBeatTimer.Q THEN
		HeartBeatStep:=0;
		HeartBeatCounts:=0;
		EmergencyStop:=1;
		HeartBeatTimer(IN:=FALSE);
	END_IF
	IF HeartBeatCounts=32767THEN
		HeartBeatCounts:=1;
	END_IF
END_IF
IF EmergencyStop=1AND((diRotateHomestep+ diRotateJogstep+diRotateMovetostep<>0)OR(diTraverseHomestep+diTraverseJogstep+diTraverseMovetostep <>0))THEN
	diRotateStopstep:=1;
	diTraverseStopstep:=2;
	diRotateHomestep:=0;
	diRotateJogstep:=0;
	diRotateMovetostep:=0;
	diTraverseHomestep:=0;
	diTraverseJogstep:=0;
	diTraverseMovetostep:=0;
	xStop2:=TRUE;
	EmergencyStop:=0;
ELSIF EmergencyStop=1AND((diRotateHomestep+ diRotateJogstep+diRotateMovetostep+diRotateStopstep=0)OR(diTraverseHomestep+diTraverseJogstep+diTraverseMovetostep+ diTraverseStopstep=0))THEN
	EmergencyStop:=0;
END_IF
IF pCanOpenNode[0].nStatus<>5 THEN(*canopen通讯异常，无法通过程序控制电机*)
	RETURN;
END_IF
fbReset1(Execute:= xReset1,pControlword:=ADR(control1));(*清除旋转部驱动器错误*)

fbReset2(Execute:= xReset2,pControlword:=ADR(control2));(*清除病床驱动器错误*)

fbPower1(Axis:=1 ,											(*大驱动器使能*)
			xPowerOn:= xPowerOn1,
			xPowerOff:= xPowerOff1,
			pControlword:=ADR(control1) ,
			pStatusword:= ADR(state1));
fbStop1(Axis:= 1,Execute:= xStop1,pControlword:= ADR(control1),pStatusword:= ADR(state1),pVelocity:=ADR(jogvel1));
fbRelMove1(Axis:= 1,Execute:= xRelativeExe1,				(*大驱动器相对位置*)
			Acceleration:= Acc,Deceleration:=Dec,
			ProfileVelocity:= diVelocity1,TargetPosition:= diPosition1,
			pControlword:= ADR(control1),pStatusword:= ADR(state1),
			pTargetPosition:= ADR(position1),pVelocityInPPmode:= ADR(velocity1));
fbVelMove1(Axis:= 1,											(*大驱动器速度*)
			Execute:= xVelocityExe1,
			Acceleration:=Acc,Deceleration:=Dec,
			Velocity_jog:= diVelocity_jog1,pVelocity:= ADR(JogVel1),
			pControlword:= ADR(control1),pStatusword:= ADR(state1));
fbPower2(Axis:= 2 ,
			xPowerOn:= xPowerOn2,
			xPowerOff:= xPowerOff2,
			pControlword:=ADR(control2) ,
			pStatusword:= ADR(state2));
fbRelMove2(Axis:= 2,
			Execute:= xRelativeExe2,
			Acceleration:= 1000000,
			Deceleration:= 1000000,
			ProfileVelocity:= diVelocity2,
			TargetPosition:= diPosition2,
			pControlword:= ADR(control2),
			pStatusword:= ADR(state2),
			pTargetPosition:= ADR(position2),
			pVelocityInPPmode:= ADR(velocity2));
fbVelMove2(Axis:= 2,
			Execute:= xVelocityExe2,
			Acceleration:= 1000000,
			Deceleration:=1800000,
			Velocity_jog:= diVelocity_jog2,
			pVelocity:= ADR(JogVel2),
			pControlword:= ADR(control2),
			pStatusword:= ADR(state2));
fbStop2(Axis:= 2,Execute:= xStop2,pControlword:= ADR(control2),pStatusword:= ADR(state2),pVelocity:=ADR(jogvel2));
END_PROGRAM

(* POU PLCOpen_CAN2.3/运动控制功能块/MC_MoveRelative, ST *)
FUNCTION_BLOCK MC_MoveRelative
(*This Function Block commands a controlled motion of a specified distance realative to the set position
at the time of the execution *)
VAR_INPUT
	Axis					: USINT;					(*Node ID*)
	Execute				: BOOL;					(*Starting Moving at rising edge*)
	Acceleration			: UDINT;					(*Acceleration of motion*)
	Deceleration			: UDINT;					(*Deceleration of motion*)
	ProfileVelocity			: UDINT;					(*Velocity of motion*)
	TargetPosition			: DINT;						(*Target position of motion*)
	pControlword			: POINTER TO UINT;		(*Adress of PDO:Controlword 0x6040*)
	pStatusword			: POINTER TO UINT;		(*Adress of PDO:Statusword 0x6041*)
	pTargetPosition		: POINTER TO DINT;		(*Adress of PDO:Target Position 0x607A*)
	pVelocityInPPmode	: POINTER TO UDINT;		(*Adress of PDO:Profile Velocity in PP mode 0x6081*)
	Timeout				: TIME:=t#1000ms;
END_VAR
VAR_OUTPUT
	Done					: BOOL;		(*Target position reached*)
	Busy					: BOOL;		(*FB is working*)
	Error					: BOOL;		(*Signals that error has occurred within the FB*)
	ErrCode				: INT;			(*0:Normal 1:Driver status error 2:Communication timeout*)
END_VAR
VAR
	RTrig:R_TRIG;
	FTrig:F_TRIG;
	SDO:SDOWrite;
	(*SDO-mode, use 16#40 FOR read-request,
		use 16#23 FOR 4-BYTE-write-request.
		use 16#27 for 3-byte...
		use 16#2B for 2-byte...
		use 16#2F for 1-byte...
		use 16#21 FOR downloading more than 4 bytes using the segmented transfer.*)
	xEnable: BOOL;
	iStep: INT;
	Timer: TON;
	i: INT;
	usiCurrentMode: USINT;
	xAxisUnderControl: BOOL;		(*indicate that the axis is controlled*)
	iIndex: INT;		(*driver index in the GLB list*)
	iAxisAmount: INT := 0;
END_VAR
RTrig(CLK:=Execute);
FTrig(CLK:=Execute);

IF RTrig.Q THEN
	xEnable:=TRUE;
	Done:=FALSE;
	Error:=FALSE;
	ErrCode:=0;
	Busy:=TRUE;
	xAxisUnderControl:=FALSE;
	iAxisAmount:=UDINT_TO_INT(g_CAN_udiStationAmount);
	iIndex:=0;
	FOR i:=1 TO iAxisAmount DO
		IF Axis=g_CAN_arAxis[i].usiAxis THEN
			usiCurrentMode:=g_CAN_arAxis[i].usiCurrentMode;
			xAxisUnderControl:=TRUE;
			iIndex:=i;
		END_IF
	END_FOR
	IF NOT xAxisUnderControl THEN
		g_CAN_udiStationAmount:=g_CAN_udiStationAmount+1;
		iIndex:=UDINT_TO_INT(g_CAN_udiStationAmount);
		g_CAN_arAxis[iIndex].usiAxis:=Axis;
		iStep:=0;
	ELSE
		IF g_CAN_arAxis[iIndex].usiCurrentMode<>1 THEN
			iStep:=0;
		ELSE
			iStep:=4;
		END_IF
	END_IF
END_IF
(*
IF FTrig.Q THEN
	xEnable:=FALSE;
	iStep:=-1;
	Busy:=FALSE;
	Done:=FALSE;
	pControlword^:=16#10F;
	SDO(xEnable:=FALSE);
	Timer(IN:=FALSE);
END_IF
*)
CASE iStep OF
0:	(*Clear alarm*)
	IF pStatusword^=0 THEN
		Error:=TRUE;
		ErrCode:=1;
		iStep:=-1;
		RETURN;
	END_IF
	pControlword^:=16#80;
	iStep:=1;

1:	(*shutdown*)
	pControlword^:=16#06;
	Timer(IN:=TRUE, PT:=TimeOut);
	IF (UINT_TO_WORD(pStatusword^) AND 16#0F)=16#01 THEN
		Timer(IN:=FALSE);
		iStep:=2;
	END_IF
	IF Timer.Q THEN
		iStep:=-1;
		Error:=TRUE;
		ErrCode:=2;
		Timer(IN:=FALSE);
		Busy:=FALSE;
	END_IF

2:	(*switch on*)
	pControlword^:=16#07;
	Timer(IN:=TRUE, PT:=TimeOut);
	IF (UINT_TO_WORD(pStatusword^) AND 16#0F)=16#03 THEN
		Timer(IN:=FALSE);
		iStep:=3;
	END_IF
	IF Timer.Q THEN
		iStep:=-1;
		Error:=TRUE;
		ErrCode:=2;
		Timer(IN:=FALSE);
		Busy:=FALSE;
	END_IF

3:	(*Set PP mode*)
	SDO(
		xEnable:=TRUE ,
		byNodeID:=Axis ,
		dwData:=1 ,
		iLength:=1 ,
		wIndex:=16#6060 ,
		bySubIndex:=0 ,
		tTimeOut:=Timeout);
	IF SDO.xError THEN
		SDO(xEnable:=FALSE);
		iStep:=-1;
		Error:=TRUE;
		ErrCode:=2;
		RETURN;
	END_IF
	IF SDO.xDone THEN
		SDO(xEnable:=FALSE);
		g_CAN_arAxis[iIndex].usiCurrentMode:=1;
		iStep:=8;
	END_IF
8:  pControlword^:=16#0F;
     istep:=4;
4:	(*Set Acc*)
	SDO(
		xEnable:=TRUE ,
		byNodeID:=Axis ,
		dwData:=UDINT_TO_DWORD(Acceleration) ,
		iLength:=4 ,
		wIndex:=16#6083 ,
		bySubIndex:=0 ,
		tTimeOut:=Timeout ,
		xDone=> ,
		xError=> ,
		iErrCode=> );
	IF SDO.xError THEN
		SDO(xEnable:=FALSE);
		iStep:=-1;
		Error:=TRUE;
		ErrCode:=2;
	END_IF
	IF SDO.xDone THEN
		SDO(xEnable:=FALSE);
		iStep:=5;
	END_IF

5:	(*Set Dec*)
	SDO(
		xEnable:=TRUE ,
		byNodeID:=Axis ,
		dwData:=UDINT_TO_DWORD(Deceleration) ,
		iLength:=4 ,
		wIndex:=16#6084 ,
		bySubIndex:=0 ,
		tTimeOut:=Timeout ,
		xDone=> ,
		xError=> ,
		iErrCode=> );
	IF SDO.xError THEN
		SDO(xEnable:=FALSE);
		iStep:=-1;
		Error:=TRUE;
		ErrCode:=2;
	END_IF
	SDO(xEnable:=FALSE);
	pTargetPosition^:=TargetPosition;
	pVelocityInPPmode^:=ProfileVelocity;
	pControlword^:=16#6F;
	iStep:=6;

(*	4:	(*Set profile velocity*)
	SDO(
		xEnable:=TRUE ,
		byNodeID:=Axis ,
		dwData:=DINT_TO_DWORD(ProfileVelocity) ,
		iLength:=4 ,
		wIndex:=16#6081 ,
		bySubIndex:=0 ,
		tTimeOut:=t#100ms ,
		xDone=> ,
		xError=> ,
		iErrCode=> );
	IF SDO.xError THEN
		SDO(xEnable:=FALSE);
		iStep:=-1;
		Error:=TRUE;
		ErrCode:=2;
	END_IF
	IF SDO.xDone THEN
		SDO(xEnable:=FALSE);
		iStep:=5;
	END_IF

5:	(*Set target position*)
	SDO(
		xEnable:=TRUE ,
		byNodeID:=Axis ,
		dwData:=DINT_TO_DWORD(TargetPosition) ,
		iLength:=4 ,
		wIndex:=16#607A ,
		bySubIndex:=0 ,
		tTimeOut:=t#100ms ,
		xDone=> ,
		xError=> ,
		iErrCode=> );
	IF SDO.xError THEN
		SDO(xEnable:=FALSE);
		iStep:=-1;
		Error:=TRUE;
		ErrCode:=2;
	END_IF
	IF SDO.xDone THEN
		SDO(xEnable:=FALSE);
		iStep:=6;
	END_IF
*)
6:	(*New setpoint*)
	pControlword^:=16#7F;
	Timer(IN:=TRUE, PT:=TimeOut);
	IF Timer.Q THEN
		iStep:=-1;
		Error:=TRUE;
		ErrCode:=1;
		Busy:=FALSE;
		Timer(IN:=FALSE);
	END_IF
	IF pStatusword^.12 THEN
		pControlword^:=16#6F;
		Timer(IN:=FALSE);
		iStep:=7;
	END_IF

7:	(*waitting for point reach*)
	IF pStatusword^.10 THEN
		iStep:=-1;
		xEnable:=FALSE;
		Done:=TRUE;
		Busy:=FALSE;
	END_IF

END_CASE
END_FUNCTION_BLOCK

(* POU PLCOpen_CAN2.3/运动控制功能块/SDOWrite, ST *)
FUNCTION_BLOCK SDOWrite
(*This FB is used for sending SDO, it will set timer for waitting answer. *)
VAR_INPUT
	xEnable			: BOOL;				(*Rising edge enable the FB to send one SDO*)
	byNodeID		: BYTE;				(*Station ID*)
	dwData			: DWORD;			(*Data to be send*)
	iLength			: INT;				(*bytes number, can be 1,2,3 or 4*)
	wIndex			: WORD;			(*index to write data*)
	bySubIndex	: BYTE;				(*subindex to write data*)
	tTimeOut		:TIME:=t#100ms;	(*after this time, if there was no answer, there will be an error code*)
END_VAR
VAR_OUTPUT
	xDone			: BOOL;			(*SDO answer received*)
	xError			: BOOL;			(*error happend*)
	iErrCode		: INT;			(*0:normal	1:timeout	2:date length error*)
END_VAR
VAR
	RTrig:R_TRIG;
	FTrig:F_TRIG;
	SDO:CanOpenSendSDO;	(*SDO-mode, use 16#40 FOR read-request,
		use 16#23 FOR 4-BYTE-write-request.
		use 16#27 for 3-byte...
		use 16#2B for 2-byte...
		use 16#2F for 1-byte...
		use 16#21 FOR downloading more than 4 bytes using the segmented transfer.*)
	iStep: INT := -1;
	byModus: BYTE := 00;
	Timer: TON;
	iRetryTime: INT := 1;		(*try to send SDO again times*)
	iRetryCount: INT := 0;		(*retry counter*)
END_VAR
RTrig(CLK:=xEnable);
FTrig(CLK:=xEnable);

IF RTrig.Q THEN
	xDone:=FALSE;
	xError:=FALSE;
	iErrCode:=0;
	CASE iLength OF
	1:
		byModus:=16#2F;
	2:
		byModus:=16#2B;
	3:
		byModus:=16#27;
	4:
		byModus:=16#23;
	ELSE
		byModus:=0;
		xError:=TRUE;
		iErrCode:=2;
		iStep:=-1;
		RETURN;
	END_CASE
	iStep:=0;
	iRetryCount:= 0;
END_IF

IF FTrig.Q THEN
	SDO(Enable:=FALSE);
	iStep:=-1;
END_IF

CASE iStep OF
0:
	SDO(
		Enable:=TRUE ,
		wDrvNr:=0 ,
		ucNodeId:=byNodeID ,
		wIndex:=wIndex ,
		bySubIndex:=bySubIndex ,
		ucModus:=byModus ,
		ucByte0:=DWORD_TO_BYTE(dwData) ,
		ucByte1:=DWORD_TO_BYTE(SHR(dwData,8)) ,
		ucByte2:=DWORD_TO_BYTE(SHR(dwData,16)),
		ucByte3:=DWORD_TO_BYTE(SHR(dwData,24)) ,
		aAbortCode:= ,
		dwDataBufferLength:= ,
		pDataBuffer:= ,
		bWaitForAnswer=> ,
		bAnswerRec=> , 
		ucAnswerBytes=> , 
		iAnswerLength=> ,
		bToggleUnequal=> , 
		bAbortRec=> ,
		aAbortRec=> ,
		dwReadDataLen=> );
	iStep:=1;
1:
	iStep:=-1;
	xDone:=TRUE;
	SDO(Enable:=FALSE);

(*	SDO();
	Timer(IN:=TRUE, PT:=tTimeOut);
	IF SDO.bAnswerRec THEN
		IF SDO.ucAnswerBytes[0]<>16#60 THEN
			iErrCode:=2;
		END_IF
		iStep:=-1;
		xDone:=TRUE;
		SDO(Enable:=FALSE);
		Timer(IN:=FALSE);
		RETURN;
	END_IF
	IF Timer.Q THEN
		iRetryCount:=iRetryCount+1;
		SDO(Enable:=FALSE);
		Timer(IN:=FALSE);
		iStep:=0;
		IF iRetryCount=iRetryTime THEN
			iStep:=-1;
			iErrCode:=1;
			xError:=TRUE;
		END_IF
	END_IF*)
END_CASE
END_FUNCTION_BLOCK

(* POU PLCOpen_CAN2.3/运动控制功能块/MC_Power, ST *)
FUNCTION_BLOCK MC_Power
(*This Function Block controls the power stage*)
VAR_INPUT
	Axis					: BYTE;
	xPowerOn				: BOOL;
	xPowerOff				: BOOL;
	(*Enable_Positive			: BOOL;			(*unimplemented*)
	Enable_Negative		: BOOL;				(*unimplemented*)*)
	pControlword			: POINTER TO UINT;
	pStatusword			: POINTER TO UINT;
END_VAR
VAR_OUTPUT
	xDone					:BOOL;
	Error					:BOOL:=FALSE;		(* Signals that Error hasoccured within Function block *)
	ErrorID					:INT;					(* Error Number *)
END_VAR
VAR
	iFunction: INT;
	iSerOnStep: INT;
	iSerOffStep: INT;

	OnRTrig: R_TRIG;
	OffRTrig: R_TRIG;
END_VAR
OnRTrig(CLK:= xPowerOn);
OffRTrig(CLK:= xPowerOff);

IF OnRTrig.Q THEN
	iFunction:=1;
	iSerOnStep:= 0;
	xDone:= FALSE;
END_IF

IF OffRTrig.Q THEN
	iFunction:=-1;
	iSerOffStep:= 0;
	xDone:= FALSE;
END_IF

CASE iFunction OF
1:
	CASE iSerOnStep OF
	0:		(*wait for driver ready*)
		(*pControlword^:=16#100;*)
		(*Timer(IN:=TRUE, PT:=t#2s);
		IF Timer.Q THEN
			iSerOnStep:=1;
			Timer(IN:=FALSE);
		END_IF*)
		IF (UINT_TO_WORD(pStatusword^) AND 16#0008) = 0 THEN
			iSerOnStep:=2;
		ELSE
			iSerOnStep:=1;
		END_IF
		(*iSerOnStep:=1;*)

	1:		(*Fault Reset*)
		pControlword^:=16#80;
		IF (UINT_TO_WORD(pStatusword^) AND 16#0008) = 0 THEN
			iSerOnStep:=2;
		END_IF

	2:		(*Shut Down*)
		pControlword^:=16#06;
		IF pStatusword^.0 AND pStatusword^.5 THEN
(*		IF (UINT_TO_WORD(pStatusword^) AND 16#FF)=16#21 THEN*)
			iSerOnStep:=3;
		END_IF

	3:		(*Switch On*)
		pControlword^:=16#07;
		IF pStatusword^.0 AND pStatusword^.5 AND pStatusword^.1 THEN
(*		IF (UINT_TO_WORD(pStatusword^) AND 16#FF)=16#23 THEN*)
			iSerOnStep:=4;
		END_IF

	4:		(*Operation Enable*)
		pControlword^:=16#0F;
		iSerOnStep:=-1;
		xDone:= TRUE;
		iFunction:=0;
	END_CASE

-1:
	CASE iSerOffStep OF
	0:		(*Fault Reset*)
		pControlword^:=16#80;
		iSerOffStep:=1;

	1:		(*Shut Down*)
		pControlword^:=16#06;
		IF NOT pStatusword^.6 THEN
			iSerOffStep:=2;
		END_IF

	2:		(*Switch On*)
		pControlword^:=16#07;
		iSerOffStep:=-1;
		xDone:= TRUE;
		iFunction:=0;
	END_CASE
END_CASE
END_FUNCTION_BLOCK

(* POU PLCOpen_CAN2.3/运动控制功能块/MC_Stop, ST *)
FUNCTION_BLOCK MC_Stop
(*This Function Block commands a controlled motion stop and transfers the axis to the state OperationEnable. It
aborts any ongoing Function Block execution. The command will be send one time. Other FB can perform any motion
on the same axis by setting the controlword.*)
VAR_INPUT
	Axis					: BYTE;		(*Node ID*)
	Execute				: BOOL;		(*Starting Moving at rising edge*)
	pControlword		: POINTER TO UINT;		(*Adress of PDO:Controlword*)
	pStatusword		: POINTER TO UINT;		(*Adress of PDO:Statusword*)
	pVelocity				: POINTER TO DINT;
END_VAR
VAR_OUTPUT
	xBusy				: BOOL;
	xDone				: BOOL;		(*Zero velocity reached*)
END_VAR
VAR

	RTrig:R_TRIG;
	FTrig:F_TRIG;
	xEnable: BOOL;
	uiTemp: UINT;
END_VAR
RTrig(CLK:= Execute);
IF RTrig.Q THEN
	xBusy:=TRUE;
	xDone:=FALSE;
END_IF

(*IF FTrig.Q THEN
	xEnable:=FALSE;
	Done:=FALSE;
END_IF*)

IF xBusy THEN
	pControlword^:=UINT_TO_WORD(pControlword^) OR 16#0100;
	xDone:= TRUE;
	xBusy:= FALSE;
	pVelocity^:=0;
(*	IF NOT pStatusword^.5 THEN
		xDone:=TRUE;
		xBusy:= FALSE;
	END_IF*)
END_IF
END_FUNCTION_BLOCK

(* POU PLCOpen_CAN2.3/运动控制功能块/MC_MoveVelocity, ST *)
FUNCTION_BLOCK MC_MoveVelocity
(*This Function Block commands a never ending controlled motion at a specified velocity.
Starting motion at rising edge, velocity can be changed anytime
another rise edge of Execute Acceleration and Deceleration*)
VAR_INPUT
	Axis					: USINT;				(*Node ID*)
	Execute				: BOOL;				(*Starting motion at rising edge, stop at falling edge*)
	Acceleration			: UDINT;				(*Value of acceleration*)
	Deceleration			: UDINT;				(*Value of deceleration*)
	Velocity_jog				: DINT;					(*Value of velocity*)
	pVelocity				: POINTER TO DINT;	(*Adress of PDO:TargetVelocity*)
	pControlword			: POINTER TO UINT;	(*Adress of PDO:Controlword*)
	pStatusword			: POINTER TO UINT;	(*Adress of PDO:Statusword*)
	Timeout				: TIME:=t#1000ms;	(*timeout for CANbus*)
END_VAR
VAR_OUTPUT
	Done					: BOOL;		(*Target velocity reached*)
	Busy					: BOOL;		(*FB is working*)
	Error					: BOOL;		(*Signals that error has occurred within the FB*)
	ErrCode				: INT;			(*0:Normal 1:Driver status error 2:Communication timeout*)
END_VAR
VAR
	RTrig:R_TRIG;
	FTrig:F_TRIG;
	ResetTrig: R_TRIG;
	SDO:SDOWrite;
	(*SDO-mode, use 16#40 FOR read-request,
		use 16#23 for 4-BYTE-write-request.
		use 16#27 for 3-byte...
		use 16#2B for 2-byte...
		use 16#2F for 1-byte...
		use 16#21 for downloading more than 4 bytes using the segmented transfer.*)
	xEnable: BOOL;
	iStep: INT:=-1;
	Timer: TON;
	i: INT;
	usiCurrentMode: USINT;
	xAxisUnderControl: BOOL;		(*indicate that the axis is controlled*)
	iIndex: INT;		(*driver index in the GLB list*)
	iAxisAmount: INT := 0;
END_VAR
RTrig(CLK:=Execute);
FTrig(CLK:=Execute);

IF RTrig.Q THEN
	xEnable:=TRUE;
	Done:=FALSE;
	Error:=FALSE;
	ErrCode:=0;
	Busy:=TRUE;
	xAxisUnderControl:=FALSE;
	iAxisAmount:=UDINT_TO_INT(g_CAN_udiStationAmount);
	iIndex:=0;
	FOR i:=1 TO iAxisAmount DO
		IF Axis=g_CAN_arAxis[i].usiAxis THEN
			usiCurrentMode:=g_CAN_arAxis[i].usiCurrentMode;
			xAxisUnderControl:=TRUE;
			iIndex:=i;
		END_IF
	END_FOR
	IF NOT xAxisUnderControl THEN
		g_CAN_udiStationAmount:=g_CAN_udiStationAmount+1;
		iIndex:=UDINT_TO_INT(g_CAN_udiStationAmount);
		g_CAN_arAxis[iIndex].usiAxis:=Axis;
		iStep:=0;
	ELSE
		IF g_CAN_arAxis[iIndex].usiCurrentMode<>2 THEN
			iStep:=0;
		ELSE
			iStep:=4;
		END_IF
	END_IF
END_IF
(*
IF FTrig.Q THEN
	xEnable:=FALSE;
	iStep:=-1;
	Busy:=FALSE;
	InVelocity:=FALSE;
	pVelocity^:=0;
	SDO(xEnable:=FALSE);
END_IF*)

CASE iStep OF
0:	(*Clear alarm*)
	IF pStatusword^=0 THEN
		Error:=TRUE;
		ErrCode:=1;
		iStep:=-1;
		RETURN;
	END_IF
	pControlword^:=16#80;
	iStep:=1;

1:	(*shutdown*)
	pControlword^:=16#06;
	Timer(IN:=TRUE, PT:=TimeOut);
	IF Timer.Q THEN
		iStep:=-1;
		Error:=TRUE;
		ErrCode:=2;
		Timer(IN:=FALSE);
		Busy:=FALSE;
	END_IF
	IF (UINT_TO_WORD(pStatusword^) AND 16#0F)=16#01 THEN
		Timer(IN:=FALSE);
		iStep:=2;
	END_IF

2:	(*switch on*)
	pControlword^:=16#07;
	Timer(IN:=TRUE, PT:=TimeOut);
	IF Timer.Q THEN
		iStep:=-1;
		Error:=TRUE;
		ErrCode:=2;
		Timer(IN:=FALSE);
		Busy:=FALSE;
	END_IF
	IF (UINT_TO_WORD(pStatusword^) AND 16#0F)=16#03 THEN
		Timer(IN:=FALSE);
		iStep:=3;
	END_IF

3:	(*Set PV mode*)
	SDO(
		xEnable:= TRUE,
		byNodeID:=Axis ,
		dwData:=3 ,
		iLength:=1 ,
		wIndex:=16#6060 ,
		bySubIndex:=0 ,
		tTimeOut:=TimeOut ,
		xDone=> ,
		xError=> ,
		iErrCode=> );
	IF SDO.xError THEN
		SDO(xEnable:=FALSE);
		iStep:=-1;
		ErrCode:=2;
	END_IF
	IF SDO.xDone THEN
		SDO(xEnable:=FALSE);
		g_CAN_arAxis[iIndex].usiCurrentMode:=2;
		iStep:=4;
	END_IF
8:  pControlword^:=16#0F;
     istep:=4;
4:	(*Set acceleration*)
	SDO(
		xEnable:= TRUE,
		byNodeID:=Axis ,
		dwData:=UDINT_TO_DWORD(Acceleration) ,
		iLength:=4 ,
		wIndex:=16#6083 ,
		bySubIndex:=0 ,
		tTimeOut:=TimeOut ,
		xDone=> ,
		xError=> ,
		iErrCode=> );
	IF SDO.xError THEN
		SDO(xEnable:=FALSE);
		iStep:=-1;
		ErrCode:=2;
	END_IF
	IF SDO.xDone THEN
		SDO(xEnable:=FALSE);
		iStep:=5;
	END_IF

5:	(*Set deceleration*)
	SDO(
		xEnable:= TRUE,
		byNodeID:=Axis ,
		dwData:=UDINT_TO_DWORD(Deceleration) ,
		iLength:=4 ,
		wIndex:=16#6084 ,
		bySubIndex:=0 ,
		tTimeOut:=TimeOut ,
		xDone=> ,
		xError=> ,
		iErrCode=> );
	IF SDO.xError THEN
		SDO(xEnable:=FALSE);
		iStep:=-1;
		ErrCode:=2;
	END_IF
	IF SDO.xDone THEN
		SDO(xEnable:=FALSE);
		iStep:=6;
		pVelocity^:=Velocity_jog;
	END_IF

6:	(*Operation enable*)
	pControlword^:=16#0F;
	Timer(IN:=TRUE, PT:=TimeOut);
	IF Timer.Q THEN
		iStep:=-1;
		Error:=TRUE;
		ErrCode:=1;
		Busy:=FALSE;
		Timer(IN:=FALSE);
	END_IF
	IF NOT pStatusword^.12 THEN
		Timer(IN:=FALSE);
		iStep:=7;
	END_IF

7:	(*Change Target velocity*)
	IF pStatusword^.10 THEN
		iStep:=-1;
		xEnable:=FALSE;
		Done:=TRUE;
		Busy:=FALSE;
	END_IF
END_CASE
END_FUNCTION_BLOCK

(* POU PLCOpen_CAN2.3/运动控制功能块/MC_Reset, ST *)
FUNCTION_BLOCK MC_Reset
VAR_INPUT
	Execute				: BOOL;				(*Starting Moving at rising edge*)
	pControlword			: POINTER TO UINT;		(*Adress of PDO:Controlword*)
END_VAR
VAR_OUTPUT
END_VAR
VAR
	RTrig: R_TRIG;
END_VAR
RTrig(CLK:= Execute);
IF RTrig.Q THEN
	pControlword^:= 16#80;
END_IF
END_FUNCTION_BLOCK

(* POU PLCOpen_CAN2.3/公式换算/ASCII_TO_STRING, ST *)
FUNCTION ASCII_TO_STRING : STRING(1) (*Character*)
VAR_INPUT
	byByte: BYTE; (*Code*)
END_VAR
VAR
	byByteTemp: BYTE;
	byDummy: BYTE:= 0; (*end of string to avoid overflow*)
	pszString: POINTER TO STRING(1);
END_VAR
(*ASCII Code -> ASCII Character*)
byByteTemp:= byByte;
pszString:= ADR(byByteTemp);
ASCII_TO_STRING:= pszString^;
END_FUNCTION

(* POU PLCOpen_CAN2.3/公式换算/GR_POS, ST *)
FUNCTION GR_POS : LREAL
VAR_INPUT
	index_velue:DINT;
	enc_velue:LREAL;
END_VAR
VAR
END_VAR
(*IF enc_velue>= index_velue AND index_velue<>0THEN
	IF (enc_velue-DINT_TO_LREAL(index_velue))<160 THEN
		GR_POS:= 355+(enc_velue-DINT_TO_LREAL(index_velue))/32;
	ELSIF (enc_velue-DINT_TO_LREAL(index_velue))=160 THEN
		GR_POS:= 0;
	ELSIF (enc_velue-DINT_TO_LREAL(index_velue))>160 THEN
		GR_POS:=(enc_velue-160-DINT_TO_LREAL(index_velue))/32;
	END_IF
ELSIF enc_velue<0 OR index_velue<0 THEN
	GR_POS:=999.9;(*编码器受干扰*)
ELSIF enc_velue>=0AND index_velue=0THEN
	GR_POS:=888.8;(*未做HOME*)
END_IF*)
IF enc_velue>= index_velue AND index_velue<>0THEN
	GR_POS:= (enc_velue-DINT_TO_LREAL(index_velue))/16;
ELSIF enc_velue<0 OR index_velue<0 THEN
	GR_POS:=999.9;(*编码器受干扰*)
ELSIF enc_velue>=0AND index_velue=0THEN
	GR_POS:=888.8;(*未做HOME*)
END_IF
END_FUNCTION

(* POU PLCOpen_CAN2.3/公式换算/LREAL_TO_LREALDOTN, ST *)
FUNCTION LREAL_TO_LREALDOTN : LREAL
VAR_INPUT
	LrIn:LREAL;
	N:INT;
END_VAR
VAR
	VarLocal: DINT;
END_VAR
VarLocal:=LREAL_TO_DINT(LrIn*EXPT(10, N));
LREAL_TO_LREALDOTN:=DINT_TO_LREAL(VarLocal)/EXPT(10, N);
END_FUNCTION

(* POU 子程序/TiltManager, ST *)
PROGRAM TiltManager
VAR
	LanNullArray,abyRecvRaw,abyRecv,HeartBeat: ARRAY [1..256] OF BYTE;
	diReceived:DINT;
	SizeOfMsg:INT;
	diStopStep,diJogStep,diMovetoStep,diHomeStep:UINT;
	str150:STRING(50):='HOME TILT;ACK@'; str151:STRING(50):='HOME TILT;UNDERWAY@'; str152:STRING(50):='HOME TILT;COMPLETED@'; str153:STRING(50):='HOME TILT;FAILED=';
	str154:STRING(50):='JOG TILT;ACK@'; str155:STRING(50):='JOG TILT;UNDERWAY@'; str156:STRING(50):='JOG TILT;COMPLETED@'; str157:STRING(50):='JOG TILT;FAILED=';
	str158:STRING(50):='MOVETO TILT;ACK@'; str159:STRING(50):='MOVETO TILT;UNDERWAY@'; str160:STRING(50):='MOVETO TILT;COMPLETED@'; str161:STRING(50):='MOVETO TILT;FAILED=';
	str162:STRING(50):='STOP TILT;ACK@'; str163:STRING(50):='STOP TILT;UNDERWAY@'; str164:STRING(50):='STOP TILT;COMPLETED@'; str165:STRING(50):='JOG TILT;STOPPED@'; str166:STRING(50):='STOP TILT;FAILED=';
	str169:STRING(50):='SET TILT;COMPLETED@'; str170:STRING(50):='SET TILT;FAILED=';
	str173:STRING(50):='RESET TILT;COMPLETED@'; str174:STRING(50):='RESET TILT;FAILED=';
	str175:STRING(50):='MOVETO TILT;STOPPED@';str176:STRING(50):='HOME TILT;STOPPED@';str177:STRING(50):='ERROR:=';
	str178:STRING(50):='JOG TILT;FAILED=Positive Limit@';str179:STRING(50):='JOG TILT;FAILED=Negative Limit@';
	i,j,k,m,SecondColonPos: INT;
	Temp,Temp1,SendTiltAngle,SendTiltSpeed: STRING;
	RTSpeed:ARRAY [1..10] OF BYTE:=16#52,16#54,16#04,16#00,16#11,16#30,16#20,16#00;
	TILTRE:ARRAY [1..7] OF BYTE:=16#52,16#45,16#00,16#00,16#FF;
	TILTRS:ARRAY [1..6] OF BYTE:=16#52,16#53,16#00,16#00,16#CD,16#9F;
	RG:ARRAY [1..6] OF BYTE:=16#52,16#47,16#F1,16#00,16#9E,16#20;
	NeedCRCBytes:ARRAY [0..15] OF WORD;
	MoveDirection,TiltSpeed:UINT;
	TargetPosition:REAL;
	ComNullArray,byMyRead:ARRAY [1..16] OF BYTE;
	TiltUseTimer1,AutoSendMsgDelay,OverZezoAngleDelay,HeartBeatTimer:TON;
	StartCheckTiltSpeed: BOOL;
	CheckTiltSpeed:READ_SKF_SPEED;
	AutoSendMsgStep:UINT:=0;
	OverZezoAngle: UINT;
	SpeedsSet1,SpeedSet2:BYTE;
	AngleWhenJogStart:REAL;
	HeartBeatStep,HeartBeatCounts: INT;
	EmergencyStop: INT;
END_VAR
IF	 Client1.diSocket <> SOCKET_INVALID THEN
	diReceived:= TcpReceiveData(Client1.diSocket, ADR(abyRecvRaw), SIZEOF(abyRecvRaw), 10);
	IF diReceived>0 THEN
		IF abyRecvRaw[1]=16#54 AND abyRecvRaw[2]=16#49 AND abyRecvRaw[3]=16#4C AND abyRecvRaw[4]=16#54 AND diReceived=24THEN
			HeartBeat:=abyRecvRaw;
			abyRecvRaw:=LanNullArray;
		ELSIF (abyRecvRaw[1]<>16#54 OR abyRecvRaw[2]<>16#49 OR abyRecvRaw[3]<>16#4COR abyRecvRaw[4]<>16#54)AND (abyRecvRaw[diReceived-5]<>16#42 OR abyRecvRaw[diReceived-4]<>16#45 OR abyRecvRaw[diReceived-3]<>16#41 OR abyRecvRaw[diReceived-2]<>16#54)THEN
			SizeOfMsg:=DINT_TO_INT(diReceived-2);
			abyRecv:=abyRecvRaw;
			abyRecvRaw:=LanNullArray;
		ELSIF abyRecvRaw[1]=16#54 AND abyRecvRaw[2]=16#49 AND abyRecvRaw[3]=16#4C AND abyRecvRaw[4]=16#54  AND diReceived<>24THEN
			FOR i:=1TO (DINT_TO_INT(diReceived)) BY 1 DO
				IF i<=22 THEN
					HeartBeat[i]:=abyRecvRaw[i];
				END_IF
				IF i>=25 THEN
					abyRecv[i-24]:=abyRecvRaw[i];
				END_IF
				IF  i=diReceived THEN
					abyRecvRaw:=LanNullArray;
				END_IF
			END_FOR
			SizeOfMsg:=DINT_TO_INT(diReceived-26);
		ELSIF (abyRecvRaw[1]<>16#54 OR abyRecvRaw[2]<>16#49 OR abyRecvRaw[3]<>16#4C OR abyRecvRaw[4]<>16#54 )AND abyRecvRaw[diReceived-5]=16#42 AND abyRecvRaw[diReceived-4]=16#45 AND abyRecvRaw[diReceived-3]=16#41 AND abyRecvRaw[diReceived-2]=16#54THEN
			FOR i:=1 TO (DINT_TO_INT(diReceived-26))  BY 1 DO
				abyRecv[i]:=abyRecvRaw[i];
			END_FOR
			FOR i:=1 TO 22 BY 1 DO
				HeartBeat[i]:=abyRecvRaw[diReceived-24+i];
			END_FOR
			SizeOfMsg:=DINT_TO_INT(diReceived-26);
			abyRecvRaw:=LanNullArray;
		END_IF
		(*Heart Beat*)
		IF HeartBeat[1]=16#54 AND HeartBeat[2]=16#49 AND HeartBeat[3]=16#4C AND HeartBeat[4]=16#54 AND HeartBeat[5]=16#4D AND HeartBeat[6]=16#61 AND  HeartBeat[7]=16#6E AND HeartBeat[8]=16#61 AND HeartBeat[9]=16#67 AND HeartBeat[10]=16#65 AND HeartBeat[11]=16#72THEN
			HeartBeatStep:=1;
			HeartBeatCounts:=HeartBeatCounts+1;
		END_IF
	(*获取版本信息*)
		IF(abyRecv[1]=86)AND(abyRecv[2]=69)AND(abyRecv[3]=82)AND(abyRecv[4]=83)AND(abyRecv[5]=73) AND(abyRecv[6]=79)AND(abyRecv[7]=78)AND(abyRecv[8]=32)AND(abyRecv[9]=84)AND(abyRecv[10]=73)AND(abyRecv[11]=76)AND(abyRecv[12]=84)THEN
			Temp:='';
			Temp:='VERSION TILT;<>@';
			TcpSendData(Client1.diSocket, ADR(Temp), LEN(Temp), 10);
			abyRecv:=LanNullArray;
		END_IF
		IF diStopStep=0 THEN
		(*Stop动作*)
			IF(abyRecv[1]=83)AND(abyRecv[2]=84)AND(abyRecv[3]=79)AND(abyRecv[4]=80)AND(abyRecv[5]=32) AND(abyRecv[6]=84)AND(abyRecv[7]=73)AND(abyRecv[8]=76) AND(abyRecv[9]=84)THEN
				TcpSendData(Client1.diSocket, ADR(str162), LEN(str162), 0);
				IF diHomeStep>0 THEN
					TcpSendData(Client1.diSocket, ADR(str176), LEN(str176), 0);
					diHomeStep:=0;
				ELSIF diMovetoStep>0 THEN
					TcpSendData(Client1.diSocket, ADR(str175), LEN(str175), 0);
					diMovetoStep:=0;
				ELSIF diJogStep>0 THEN
					TcpSendData(Client1.diSocket, ADR(str165), LEN(str165), 0);
					diJogStep:=0;
				END_IF
				TiltUseTimer1(IN:=FALSE);
				OverZezoAngleDelay(IN:=FALSE);
				StartCheckTiltSpeed:=FALSE;
				IF OverZezoAngle=1 THEN
					OverZezoAngle:=0;
				END_IF
				diStopStep:=1;
				abyRecv:=LanNullArray;
			ELSIF (diHomeStep+ diJogStep+diMovetoStep)=0  THEN
		(*Home动作*)
				IF(abyRecv[1]=72)AND(abyRecv[2]=79)AND(abyRecv[3]=77)AND(abyRecv[4]=69)AND(abyRecv[5]=32 ) AND(abyRecv[6]=84)AND(abyRecv[7]=73)AND(abyRecv[8]=76)AND(abyRecv[9]=84) THEN
					TcpSendData(Client1.diSocket, ADR(str150), LEN(str150), 0);
					TcpSendData(Client1.diSocket, ADR(str151), LEN(str151), 0);
					Temp1:='';
					FOR j:=1 TO SizeOfMsg DO
						Temp1:=CONCAT(Temp1,ASCII_TO_STRING(abyRecv[j]));
					END_FOR
					IF Move_Angle >+0.3THEN
						IF Move_Angle >=0.3AND Move_Angle <+1 THEN
							RTSpeed[7]:=40;RTSpeed[8]:=00;MoveDirection:=0;diHomeStep:=1;
						ELSIF Move_Angle >=+1 THEN
							RTSpeed[7]:=40;RTSpeed[8]:=00;MoveDirection:=0;diHomeStep:=1;
						END_IF
					ELSIF Move_Angle <-0.3 THEN
						IF Move_Angle <-0.3AND Move_Angle >-1 THEN
							RTSpeed[7]:=40;RTSpeed[8]:=00;MoveDirection:=1;diHomeStep:=1;
						ELSIF  Move_Angle <=-1 THEN
							RTSpeed[7]:=40;RTSpeed[8]:=00;MoveDirection:=1;diHomeStep:=1;
						END_IF
					ELSIF Move_Angle >=(-0.3)AND Move_Angle <=(+0.3) THEN
						diHomeStep:=7;
					END_IF
					abyRecv:=LanNullArray;
		(*Jog动作*)
				ELSIF(abyRecv[1]=74)AND(abyRecv[2]=79)AND(abyRecv[3]=71)AND(abyRecv[4]=32)AND(abyRecv[5]=84) AND(abyRecv[6]=73)AND(abyRecv[7]=76)AND(abyRecv[8]=84) THEN
					TcpSendData(Client1.diSocket, ADR(str154), LEN(str154), 10);
					TcpSendData(Client1.diSocket, ADR(str155), LEN(str155), 10);
					Temp1:='';
					FOR j:=1 TO SizeOfMsg DO
						Temp1:=CONCAT(Temp1,ASCII_TO_STRING(abyRecv[j]));
					END_FOR
					IF  abyRecv[SizeOfMsg]=16#30 THEN
						MoveDirection:=0;
					ELSIF abyRecv[SizeOfMsg]=16#31 THEN
						MoveDirection:=1;
					END_IF
					IF STRING_TO_UINT (DELETE(DELETE(Temp1,8,(SizeOfMsg-7)),16,1))<100THEN
						RTSpeed[7]:=STRING_TO_BYTE (DELETE(DELETE(Temp1,8,(SizeOfMsg-7)),16,1));
						RTSpeed[8]:=16#00;
						SpeedsSet1:=RTSpeed[7];
						SpeedSet2:=RTSpeed[8];
					ELSIF STRING_TO_UINT (DELETE(DELETE(Temp1,8,(SizeOfMsg-7)),16,1))>=100THEN
						RTSpeed[7]:=16#00;
						RTSpeed[8]:=16#01;
						SpeedsSet1:=RTSpeed[7];
						SpeedSet2:=RTSpeed[8];
					END_IF
					AngleWhenJogStart:=Move_Angle;
					diJogStep:=1;
					abyRecv:=LanNullArray;
			(*Moveto动作*)
				ELSIF(abyRecv[1]=77)AND(abyRecv[2]=79)AND(abyRecv[3]=86)AND(abyRecv[4]=69)AND(abyRecv[5]=84) AND(abyRecv[6]=79)AND(abyRecv[7]=32)AND(abyRecv[8]=84) AND(abyRecv[9]=73)AND(abyRecv[10]=76)AND(abyRecv[11]=84)THEN
					TcpSendData(Client1.diSocket, ADR(str158), LEN(str158), 10);
					TcpSendData(Client1.diSocket, ADR(str159), LEN(str159), 10);
					Temp1:='';
					FOR j:=1 TO SizeOfMsg DO
						Temp1:=CONCAT(Temp1,ASCII_TO_STRING(abyRecv[j]));
					END_FOR
					FOR k:=1 TO SizeOfMsg DO
						IF abyRecv[k]=16#41THEN
							SecondColonPos:=k;
						END_IF
					END_FOR
					IF STRING_TO_UINT(DELETE((DELETE(Temp1,(SizeOfMsg-SecondColonPos+2),SecondColonPos-1)),19,1))<100 THEN
						RTSpeed[7]:=STRING_TO_BYTE (DELETE((DELETE(Temp1,(SizeOfMsg-SecondColonPos+2),SecondColonPos-1)),19,1));
						RTSpeed[8]:=16#00;
					ELSIF STRING_TO_UINT(DELETE((DELETE(Temp1,(SizeOfMsg-SecondColonPos+2),SecondColonPos-1)),19,1))>=100 THEN
						RTSpeed[7]:=16#00;
						RTSpeed[8]:=16#01;
					END_IF
					IF STRING_TO_REAL(DELETE(Temp1,SecondColonPos+5,1))>Move_Angle THEN
						MoveDirection:=1;diMovetoStep:=1;
					ELSIF STRING_TO_REAL(DELETE(Temp1,(SecondColonPos+5),1))<Move_Angle THEN
						MoveDirection:=0;diMovetoStep:=1;
					ELSIF ABS(STRING_TO_REAL(DELETE(Temp1,(SecondColonPos+5),1))-Move_Angle)<(+0.5) THEN
						diMovetoStep:=4;
					END_IF
					TargetPosition:=STRING_TO_REAL (DELETE(Temp1,(SecondColonPos+5),1));
					abyRecv:=LanNullArray;
				END_IF
			END_IF
		END_IF
	ELSIF diReceived<0 THEN
		CloseSocket(ADR(Client1.diSocket));
		Client1.stIPAddress:= '';
		AutoSendMsgDelay(IN:=FALSE);
	END_IF
	IF AutoSendMsgStep=0 THEN
		AutoSendMsgDelay(IN:=TRUE,PT:=t#500ms);
		IF AutoSendMsgDelay.Q THEN
			AutoSendMsgStep:=1;
			AutoSendMsgDelay(IN:=FALSE);
		END_IF
	END_IF
	IF AutoSendMsgStep=1 THEN
		SendTiltAngle:=CONCAT(CONCAT('GET TILT;COMPLETED;ANGLE=',LREAL_TO_STRING(LREAL_TO_LREALDOTN(Move_Angle,3))),'@');
		IF diJogStep<>0 THEN
			SendTiltSpeed:=CONCAT(CONCAT('GET TILT;COMPLETED;SPEED=',UINT_TO_STRING(TiltSpeed)),'@');
			TcpSendData(Client1.diSocket, ADR(SendTiltSpeed), LEN(SendTiltSpeed), 0);
		END_IF
		TcpSendData(Client1.diSocket, ADR(SendTiltAngle), LEN(SendTiltAngle), 0);
		AutoSendMsgStep:=0;
	END_IF
END_IF
IF HeartBeatCounts>0 THEN
	HeartBeatTimer(IN:=TRUE,PT:=t#2s);
	IF HeartBeatStep=1 THEN
		HeartBeat:=LanNullArray;
		HeartBeatTimer(IN:=FALSE);
		EmergencyStop:=0;
		HeartBeatStep:=0;
	END_IF
	IF HeartBeatTimer.Q THEN
		HeartBeatStep:=0;
		HeartBeatCounts:=0;
		EmergencyStop:=1;
		HeartBeatTimer(IN:=FALSE);
	END_IF
	IF HeartBeatCounts=32767THEN
		HeartBeatCounts:=1;
	END_IF
END_IF
IF EmergencyStop=1AND(diHomestep+ diJogstep+diMovetostep<>0)THEN
	diStopstep:=2;
	diHomestep:=0;
	diJogstep:=0;
	diMovetostep:=0;
	StartCheckTiltSpeed:=FALSE;
	EmergencyStop:=0;
ELSIF EmergencyStop=1AND(diHomestep+ diJogstep+diMovetostep+diStopStep=0)THEN
	EmergencyStop:=0;
END_IF
CASE  diHomeStep OF
1:
	FOR m:=1 TO 8 DO
		NeedCRCBytes[m]:=BYTE_TO_WORD(RTSpeed[m]);
	END_FOR
	RTSpeed[9]:=WORD_TO_BYTE(CRC(NeedCRCBytes,8)MOD 256);
	RTSpeed[10]:=WORD_TO_BYTE(CRC(NeedCRCBytes,8)/ 256);
	SysComWrite(ComHandle, ADR(RTSpeed), 10, 0);
	diHomeStep:=2;
2:
	IF  byRead[1]=16#52 AND  byRead[2]=16#54 THEN
		byMyRead:=byRead;
		byRead:=ComNullArray;
	END_IF
	IF byMyRead[1]=16#52 AND  byMyRead[2]=16#54 AND  byMyRead[3]=16#06 THEN
		diHomeStep:=3;
		byMyRead:=ComNullArray;
	ELSIF byMyRead[1]=16#52 AND  byMyRead[2]=16#54 AND  byMyRead[3]<>16#06 THEN
		diHomeStep:=100;
	END_IF
3:
	TILTRE[4]:=UINT_TO_BYTE(MoveDirection+1);(*判断机架位置,确定运动方向*)
	FOR m:=1 TO 5 DO
		NeedCRCBytes[m]:=BYTE_TO_WORD(TILTRE[m]);
	END_FOR
	TILTRE[6]:=WORD_TO_BYTE(CRC(NeedCRCBytes,5)MOD 256);
	TILTRE[7]:=WORD_TO_BYTE(CRC(NeedCRCBytes,5)/ 256);
	SysComWrite(ComHandle, ADR(TILTRE), 7, 0);
	diHomeStep:=4;
4:	(*如果HOMETILT=2超过3秒，则未接收到回码，RS232通讯出错*)
	IF  byRead[1]=16#52 AND  byRead[2]=16#45 THEN
		byMyRead:=byRead;
		byRead:=ComNullArray;
	END_IF
	IF  byMyRead[1]=16#52 AND  byMyRead[2]=16#45 AND  byMyRead[3]=16#06 THEN
		diHomeStep:=5;
		byMyRead:=ComNullArray;
	ELSIF byMyRead[1]=16#52 AND  byMyRead[2]=16#45 AND byMyRead[3]<>16#06THEN
		diHomeStep:=100;
	END_IF
5:
	IF ABS(Move_Angle)<(+0.5)  THEN (* 判断机架位置，运动到0°后发送RS指令*)
		SysComWrite(ComHandle, ADR(TILTRS), 6, 0);
		diHomeStep:=6;
	END_IF
6:
	IF  byRead[1]=16#52 AND  byRead[2]=16#53 THEN
		byMyRead:=byRead;
		byRead:=ComNullArray;
	END_IF
	IF  byMyRead[1]=16#52 AND  byMyRead[2]=16#53 AND  byMyRead[3]=16#06  THEN
		diHomeStep:=7;
		byMyRead:=ComNullArray;
	ELSIF byMyRead[1]=16#52 AND  byMyRead[2]=16#53 AND  byMyRead[3]<>16#06 THEN
		diHomeStep:=100;
	END_IF
7..8:
	TiltUseTimer1(IN:=TRUE,PT:=T#300ms);
	IF TiltUseTimer1.Q THEN
		IF diHomeStep=7 THEN
			TcpSendData(Client1.diSocket, ADR(str152), LEN(str152), 10);
		ELSIF	diHomeStep=8 THEN
			TcpSendData(Client1.diSocket, ADR(str153), LEN(str153), 10);
		END_IF
		diHomeStep:=0;
		TiltUseTimer1(IN:=FALSE);
	END_IF
100:
	SysComWrite(ComHandle, ADR(TILTRS), 6, 0);
	diHomeStep:=8;
END_CASE

CASE diJogStep OF
1:	IF OverZezoAngle=1 THEN
		RTSpeed[7]:=SpeedsSet1;
		RTSpeed[8]:=SpeedSet2;
	END_IF
	FOR m:=1 TO 8 DO
		NeedCRCBytes[m]:=BYTE_TO_WORD(RTSpeed[m]);
	END_FOR
	RTSpeed[9]:=WORD_TO_BYTE(CRC(NeedCRCBytes,8)MOD 256);
	RTSpeed[10]:=WORD_TO_BYTE(CRC(NeedCRCBytes,8)/ 256);
	SysComWrite(ComHandle, ADR(RTSpeed), 10, 0);
	diJogStep:=2;
2:
	IF  byRead[1]=16#52 AND  byRead[2]=16#54 THEN
		byMyRead:=byRead;
		byRead:=ComNullArray;
	END_IF
	IF byMyRead[1]=16#52 AND byMyRead[2]=16#54 AND byMyRead[3]=16#06  THEN
		diJogStep:=3;
		byMyRead:=ComNullArray;
	ELSIF byMyRead[1]=16#52 AND byMyRead[2]=16#54 AND byMyRead[3]<>16#06 THEN
		diJogStep:=100;
	END_IF
3:
	TILTRE[4]:= UINT_TO_BYTE (MoveDirection+1);
	FOR m:=1 TO 5 DO
		NeedCRCBytes[m]:=BYTE_TO_WORD(TILTRE[m]);
	END_FOR
	TILTRE[6]:=WORD_TO_BYTE(CRC(NeedCRCBytes,5)MOD 256);
	TILTRE[7]:=WORD_TO_BYTE(CRC(NeedCRCBytes,5)/ 256);
	SysComWrite(ComHandle, ADR(TILTRE), 7, 0);
	StartCheckTiltSpeed:=TRUE;
	diJogStep:=4;
4:
	IF  byRead[1]=16#52 AND  byRead[2]=16#45 THEN
		byMyRead:=byRead;
		byRead:=ComNullArray;
	END_IF
	IF byMyRead[1]=16#52 AND byMyRead[2]=16#45 AND byMyRead[3]=16#06 THEN
		diJogStep:=5;
		byMyRead:=ComNullArray;
	ELSIF byMyRead[1]=16#52 AND byMyRead[2]=16#45 AND byMyRead[3]<>16#06THEN
		diJogStep:=100;
	END_IF
5:	IF (ABS(RTSpeed[7]+100*RTSpeed[8]-TiltSpeed))<5 THEN
		TiltUseTimer1(IN:=TRUE,PT:=T#300ms);
		IF TiltUseTimer1.Q THEN
			diJogStep:=6;
   			StartCheckTiltSpeed:=FALSE;
			TcpSendData(Client1.diSocket, ADR(str156), LEN(str156), 10);
			TiltUseTimer1(IN:=FALSE);
		END_IF
	END_IF
7,8,14:
	SysComWrite(ComHandle, ADR(TILTRS), 6, 0);
	IF diJogStep=7 THEN
		diJogStep:=9;
	ELSIF  diJogStep=8 THEN
		diJogStep:=10;
	ELSIF diJogStep=14 THEN
		diJogStep:=15;
	END_IF
9,10,15:
	IF  byRead[1]=16#52 AND  byRead[2]=16#53 THEN
		byMyRead:=byRead;
		byRead:=ComNullArray;
	END_IF
	IF  byMyRead[1]=16#52 AND byMyRead[2]=16#53 AND  byMyRead[3]=16#06 THEN
		byMyRead:=ComNullArray;
		IF diJogStep=9 THEN
			diJogStep:=11;
		ELSIF  diJogStep=10 THEN
			diJogStep:=12;
		ELSIF diJogStep=15 THEN
			diJogStep:=16;
		END_IF
	ELSIF  byMyRead[1]=16#52 AND byMyRead[2]=16#53 AND byMyRead[3]<>16#06 THEN
		diJogStep:=100;
	END_IF
11..12:
	IF diJogStep=11 THEN
		TcpSendData(Client2.diSocket, ADR(str178), LEN(str178), 10);
		diJogStep:=0;
	ELSIF diJogStep=12 THEN
		TcpSendData(Client2.diSocket, ADR(str179), LEN(str179), 10);
		diJogStep:=0;
	END_IF
13:
	TiltUseTimer1(IN:=TRUE,PT:=T#300ms);
	IF TiltUseTimer1.Q THEN
		diJogStep:=0;
		StartCheckTiltSpeed:=FALSE;
		TcpSendData(Client1.diSocket, ADR(str157), LEN(str157), 10);
		TiltUseTimer1(IN:=FALSE);
	END_IF
16:	OverZezoAngleDelay(IN:=TRUE,PT:=t#2s);
	IF OverZezoAngleDelay.Q THEN
		diJogStep:=1;
		OverZezoAngleDelay(IN:=FALSE);
	END_IF
100:
	SysComWrite(ComHandle, ADR(TILTRS), 6, 0);
	diJogStep:=13;
END_CASE
IF diJogStep>0 AND diJogStep<=6  AND MoveDirection=1THEN(*软件限位，JOG动作不得超过±30°*)
	IF Move_Angle>=30THEN
		diJogStep:=7;
	END_IF
ELSIF diJogStep>0AND diJogStep<=6 AND MoveDirection=0 THEN
	IF Move_Angle<=(-30) THEN
		diJogStep:=8;
	END_IF
END_IF
IF diJogStep>0 AND OverZezoAngle=0 AND (ABS(AngleWhenJogStart)>0.3)THEN
	IF ABS(Move_Angle)<0.2 THEN;
		OverZezoAngle:=1;
		diJogStep:=14;
	END_IF
END_IF

CASE diMovetoStep OF
1:
	FOR m:=1 TO 8 DO
		NeedCRCBytes[m]:=BYTE_TO_WORD(RTSpeed[m]);
	END_FOR
	RTSpeed[9]:=WORD_TO_BYTE(CRC(NeedCRCBytes,8)MOD 256);
	RTSpeed[10]:=WORD_TO_BYTE(CRC(NeedCRCBytes,8)/ 256);
	SysComWrite(ComHandle, ADR(RTSpeed), 10, 0);
	diMovetoStep:=2;
2:
	IF  byRead[1]=16#52 AND  byRead[2]=16#54 THEN
		byMyRead:=byRead;
		byRead:=ComNullArray;
	END_IF
	IF byMyRead[1]=16#52 AND  byMyRead[2]=16#54 AND  byMyRead[3]=16#06 THEN
		byMyRead:=ComNullArray;
		diMovetoStep:=3;
	ELSIF byMyRead[1]=16#52 AND  byMyRead[2]=16#54 AND byMyRead[3]<>16#06 THEN
		diMovetoStep:=100;
	END_IF
3:
	TILTRE[4]:=UINT_TO_BYTE(MoveDirection+1);
	FOR m:=1 TO 5 DO
		NeedCRCBytes[m]:=BYTE_TO_WORD(TILTRE[m]);
	END_FOR
	TILTRE[6]:=WORD_TO_BYTE(CRC(NeedCRCBytes,5)MOD 256);
	TILTRE[7]:=WORD_TO_BYTE(CRC(NeedCRCBytes,5)/ 256);
	SysComWrite(ComHandle, ADR(TILTRE), 7, 0);
	diMovetoStep:=4;
4:
	IF  byRead[1]=16#52 AND  byRead[2]=16#45 THEN
		byMyRead:=byRead;
		byRead:=ComNullArray;
	END_IF
	IF  byMyRead[1]=16#52 AND  byMyRead[2]=16#45 AND  byMyRead[3]=16#06  THEN
		diMovetoStep:=5;
		byMyRead:=ComNullArray;
	ELSIF byMyRead[1]=16#52 AND  byMyRead[2]=16#45 AND byMyRead[3]<>16#06 THEN
		diMovetoStep:=100;
	END_IF
5:
	IF ABS(TargetPosition-Move_Angle)<+0.5  THEN                                                          (* 判断外部编码器，到位后发送stop指令*)
		diMovetoStep:=6;
	END_IF
6:
	SysComWrite(ComHandle, ADR(TILTRS), 6, 0);
	diMovetoStep:=7;
7:
	IF  byRead[1]=16#52 AND  byRead[2]=16#53 THEN
		byMyRead:=byRead;
		byRead:=ComNullArray;
	END_IF
	IF  byMyRead[1]=16#52 AND  byMyRead[2]=16#53 AND  byMyRead[3]=16#06 THEN
		diMovetoStep:=8;
		byMyRead:=ComNullArray;
	ELSIF byMyRead[1]=16#52 AND  byMyRead[2]=16#53 AND  byMyRead[3]<>16#06THEN
		diMovetoStep:=100;
	END_IF
8..9:
	TiltUseTimer1(IN:=TRUE,PT:=T#300ms);
	IF TiltUseTimer1.Q THEN
		IF	diMovetoStep=8 THEN
			TcpSendData(Client1.diSocket, ADR(str160), LEN(str160), 10);
		ELSIF diMovetoStep=9 THEN
			TcpSendData(Client1.diSocket, ADR(str161), LEN(str161), 10);
		END_IF
		diMovetoStep:=0;
		TiltUseTimer1(IN:=FALSE);
	END_IF
100:
	SysComWrite(ComHandle, ADR(TILTRS), 6, 0);
	diMovetoStep:=9;
END_CASE
CASE diStopStep OF
1:	TiltUseTimer1(IN:=TRUE,PT:=T#300ms);
	IF TiltUseTimer1.Q THEN
		TcpSendData(Client1.diSocket, ADR(str163), LEN(str163), 10);
		diStopStep:=2;
		TiltUseTimer1(IN:=FALSE);
	END_IF
2:
	SysComWrite(ComHandle, ADR(TILTRS), 6, 0);
	diStopStep:=3;
3:
	IF  byRead[1]=16#52 AND  byRead[2]=16#53 THEN
		byMyRead:=byRead;
		byRead:=ComNullArray;
	END_IF
	IF byMyRead[1]=16#52 AND byMyRead[2]=16#53 AND byMyRead[3]=16#06 THEN
		diStopStep:=4;
		byMyRead:=ComNullArray;
	ELSIF byMyRead[1]=16#52 AND byMyRead[2]=16#53 AND  byMyRead[3]<>16#06 THEN
		diStopStep:=100;
	END_IF
4..5:
	TiltUseTimer1(IN:=TRUE,PT:=T#300ms);
	IF TiltUseTimer1.Q THEN
		IF diStopStep=4 THEN
			TcpSendData(Client1.diSocket, ADR(str164), LEN(str164), 10);
		ELSIF	diStopStep=5 THEN
			TcpSendData(Client1.diSocket, ADR(str166), LEN(str166), 10);
		END_IF
		diStopStep:=0;
		TiltUseTimer1(IN:=FALSE);
	END_IF
100:
	SysComWrite(ComHandle, ADR(TILTRS), 6, 5);
	diStopStep:=5;
END_CASE
CheckTiltSpeed(Execute:=StartCheckTiltSpeed, recieve:=byRead,RG:=RG,SPEED=>TiltSpeed);(*推杆实时速度*)
END_PROGRAM

(* POU PLCOpen_CAN2.3/串口通讯/READ_SKF_SPEED, ST *)
FUNCTION_BLOCK READ_SKF_SPEED
VAR_INPUT
	Execute:BOOL;
	recieve:ARRAY [1..16] OF BYTE;
	WAIT_RC:BOOL;
	RG:ARRAY [1..6] OF BYTE;
END_VAR

VAR_OUTPUT
	SPEED:UINT;
END_VAR

VAR
	Timer1:TON;
	Step:UINT:=0;
END_VAR
CASE	Step OF
0:	IF Execute THEN
		Step:=1;
	ELSE
		Step:=0;
	END_IF
1:	Timer1(IN:=TRUE,PT:=t#100ms);
	IF Timer1.Q AND (WAIT_RC=FALSE) THEN
		SysComWrite(ComHandle, ADR(RG), 6, 0);
		Step:=2;
		Timer1(IN:=FALSE,PT:=t#100ms);
	END_IF
2:	IF  recieve[1]=16#52 AND  recieve[2]=16#47 AND  recieve[3]=16#06  THEN
		SPEED:=BYTE_TO_UINT (recieve[6]);
		Step:=1;
	ELSE
		Step:=1;
	END_IF
END_CASE
IF Execute=FALSE THEN
	Step:=0;
	Timer1(IN:=FALSE,PT:=t#100ms);
END_IF
END_FUNCTION_BLOCK

(* POU PLCOpen_CAN2.3/公式换算/CRC, ST *)
FUNCTION CRC : WORD
VAR_INPUT
	datain:ARRAY [0..15] OF WORD;
	length:UINT;
END_VAR
VAR
	i,j:UINT;
	point:UINT:=128;
END_VAR
CRC:=0;
FOR i:=1 TO length DO
	point:=128;
	WHILE(point>0) DO
		IF(CRC AND 16#8000 )<>0 THEN
			CRC:=(CRC*2 ) AND 16#FFFF;
			CRC:=  CRC  XOR 16#1021;
		 ELSE
			CRC:=  (CRC*2) AND 16#FFFF;
		 END_IF;
		IF(datain[i] AND UINT_TO_WORD(point))<>0 THEN
			CRC:=  CRC  XOR 16#1021;
		END_IF
		point:=point/2;
	END_WHILE
END_FOR
END_FUNCTION

(* POU 子程序/LiftManager, ST *)
PROGRAM LiftManager
VAR
	LanNullArray,abyRecvRaw,abyRecv,HeartBeat: ARRAY [1..256] OF BYTE;
	diReceived:DINT;
	SizeOfMsg:INT;
	diStopStep,diJogStep,diMovetoStep,diHomeStep:UINT;
	str100:STRING(50):='HOME LIFT;ACK@'; str101:STRING(50):='HOME LIFT;UNDERWAY@'; str102:STRING(50):='HOME LIFT;COMPLETED@'; str103:STRING(50):='HOME LIFT;FAILED=';
	str104:STRING(50):='JOG LIFT;ACK@'; str105:STRING(50):='JOG LIFT;UNDERWAY@'; str106:STRING(50):='JOG LIFT;COMPLETED@'; str107:STRING(50):='JOG LIFT;FAILED=';
	str108:STRING(50):='MOVETO LIFT;ACK@'; str109:STRING(50):='MOVETO LIFT;UNDERWAY@'; str110:STRING(50):='MOVETO LIFT;COMPLETED@'; str111:STRING(50):='MOVETO LIFT;FAILED=';
	str112:STRING(50):='STOP LIFT;ACK@'; str113:STRING(50):='STOP LIFT;UNDERWAY@'; str114:STRING(50):='STOP LIFT;COMPLETED@'; str115:STRING(50):='JOG LIFT;STOPPED@'; str116:STRING(50):='STOP LIFT;FAILED=';
	str123:STRING(50):='RESET LIFT;COMPLETED@'; str124:STRING(50):='RESET LIFT;FAILED=';
	str125:STRING(50):='MOVETO LIFT;STOPPED@';str126:STRING(50):='HOME LIFT;STOPPED@';
	str127:STRING(50):='JOG LIFT;FAILED=Up Limit@';str128:STRING(50):='JOG LIFT;FAILED=Down Limit@';
	i,j,k,m,SecondColonPos,SendTimes: INT;
	Temp,Temp1,SendLiftHeight,SendLiftSpeed: STRING;
	NeedCRCBytes:ARRAY [0..15] OF WORD;
	ComNullArray,byMyRead:ARRAY [1..16] OF BYTE;
	LIFTRE:ARRAY [1..7] OF BYTE:=16#52,16#45,16#01,16#00,16#FF;
	LIFTRS:ARRAY [1..6] OF BYTE:=16#52,16#53,16#01,16#00,16#FC,16#AC;
	RTSpeed:ARRAY [1..10] OF BYTE:=16#52,16#54,16#04,16#00,16#12,16#30,16#20,16#00;
	RG:ARRAY [1..6] OF BYTE:=16#52,16#47,16#F2,16#00,16#CD,16#75;
	Dir:UINT;
	LiftUseTimer1,LiftUseTimer2,AutoSendMsgDelay,HeartBeatTimer:TON;
	TargetPosition:REAL;
	StartCheckSpeed: BOOL;
	CheckLiftSpeed:READ_SKF_SPEED;
	Vert_Limit_Up,Vert_Limit_Down:UINT;
	AutoSendMsgStep:UINT:=0;
	HeartBeatStep,HeartBeatCounts: INT;
	EmergencyStop: INT;

	myStartLiftDelta : REAL:= 0;
	mykPostionAllowError : REAL:= 2;

END_VAR
IF	 Client2.diSocket <> SOCKET_INVALID THEN
	diReceived:= TcpReceiveData(Client2.diSocket, ADR(abyRecvRaw), SIZEOF(abyRecvRaw), 10);
	IF diReceived>0 THEN
		IF abyRecvRaw[1]=16#4C AND abyRecvRaw[2]=16#49 AND abyRecvRaw[3]=16#46 AND abyRecvRaw[4]=16#54 AND diReceived=24THEN
			HeartBeat:=abyRecvRaw;
			abyRecvRaw:=LanNullArray;
		ELSIF (abyRecvRaw[1]<>16#4C OR abyRecvRaw[2]<>16#49 OR abyRecvRaw[3]<>16#46OR abyRecvRaw[4]<>16#54)AND (abyRecvRaw[diReceived-5]<>16#42 OR abyRecvRaw[diReceived-4]<>16#45 OR abyRecvRaw[diReceived-3]<>16#41 OR abyRecvRaw[diReceived-2]<>16#54)THEN
			SizeOfMsg:=DINT_TO_INT(diReceived-2);
			abyRecv:=abyRecvRaw;
			abyRecvRaw:=LanNullArray;
		ELSIF abyRecvRaw[1]=16#4C AND abyRecvRaw[2]=16#49 AND abyRecvRaw[3]=16#46 AND abyRecvRaw[4]=16#54  AND diReceived<>24THEN
			FOR i:=1TO (DINT_TO_INT(diReceived)) BY 1 DO
				IF i<=22 THEN
					HeartBeat[i]:=abyRecvRaw[i];
				END_IF
				IF i>=25 THEN
					abyRecv[i-24]:=abyRecvRaw[i];
				END_IF
				IF  i=diReceived THEN
					abyRecvRaw:=LanNullArray;
				END_IF
			END_FOR
			SizeOfMsg:=DINT_TO_INT(diReceived-26);
		ELSIF (abyRecvRaw[1]<>16#4C OR abyRecvRaw[2]<>16#49 OR abyRecvRaw[3]<>16#46 OR abyRecvRaw[4]<>16#54 )AND abyRecvRaw[diReceived-5]=16#42 AND abyRecvRaw[diReceived-4]=16#45 AND abyRecvRaw[diReceived-3]=16#41 AND abyRecvRaw[diReceived-2]=16#54THEN
			FOR i:=1 TO (DINT_TO_INT(diReceived-26))  BY 1 DO
				abyRecv[i]:=abyRecvRaw[i];
			END_FOR
			FOR i:=1 TO 22 BY 1 DO
				HeartBeat[i]:=abyRecvRaw[diReceived-24+i];
			END_FOR
			SizeOfMsg:=DINT_TO_INT(diReceived-26);
			abyRecvRaw:=LanNullArray;
		END_IF
		(*Heart Beat*)
		IF HeartBeat[1]=16#4C AND HeartBeat[2]=16#49 AND HeartBeat[3]=16#46 AND HeartBeat[4]=16#54 AND HeartBeat[5]=16#4D AND HeartBeat[6]=16#61 AND  HeartBeat[7]=16#6E AND HeartBeat[8]=16#61 AND HeartBeat[9]=16#67 AND HeartBeat[10]=16#65 AND HeartBeat[11]=16#72THEN
			HeartBeatStep:=1;
			HeartBeatCounts:=HeartBeatCounts+1;
		END_IF
	(*获取版本信息*)
		IF(abyRecv[1]=86)AND(abyRecv[2]=69)AND(abyRecv[3]=82)AND(abyRecv[4]=83)AND(abyRecv[5]=73) AND(abyRecv[6]=79)AND(abyRecv[7]=78)AND(abyRecv[8]=32)AND(abyRecv[9]=76)AND(abyRecv[10]=73)AND(abyRecv[11]=70)AND(abyRecv[12]=84)THEN
			Temp:='';
			Temp:='VERSION LIFT;<>@';
			TcpSendData(Client2.diSocket, ADR(Temp), LEN(Temp), 10);
			abyRecv:=LanNullArray;
		END_IF
		IF	diStopStep=0 THEN
		(*STOP*)
			IF(abyRecv[1]=83)AND(abyRecv[2]=84)AND(abyRecv[3]=79)AND(abyRecv[4]=80)AND(abyRecv[5]=32) AND(abyRecv[6]=76)AND(abyRecv[7]=73)AND(abyRecv[8]=70) AND(abyRecv[9]=84)THEN
				TcpSendData(Client2.diSocket, ADR(str112), LEN(str112), 10);
				IF diHomeStep>0 THEN
					TcpSendData(Client2.diSocket, ADR(str126), LEN(str126), 10);
					diHomeStep:=0;
				ELSIF diMovetoStep>0 THEN
					TcpSendData(Client2.diSocket, ADR(str125), LEN(str125), 10);
					diMovetoStep:=0;
				ELSIF diJogStep>0 THEN
					TcpSendData(Client2.diSocket, ADR(str115), LEN(str115), 10);
					diJogStep:=0;
				END_IF
				LiftUseTimer1(IN:=FALSE);
				StartCheckSpeed:=FALSE;
				diStopStep:=1;
				abyRecv:=LanNullArray;
			ELSIF	(diHomeStep+ diJogStep+ diMovetoStep)=0  THEN
		(*HOME动作*)
				 IF(abyRecv[1]=72)AND(abyRecv[2]=79)AND(abyRecv[3]=77)AND(abyRecv[4]=69)AND(abyRecv[5]=32 ) AND(abyRecv[6]=76)AND(abyRecv[7]=73)AND(abyRecv[8]=70)AND(abyRecv[9]=84) THEN
					TcpSendData(Client2.diSocket, ADR(str100), LEN(str100), 0);
					TcpSendData(Client2.diSocket, ADR(str101), LEN(str101), 0);
					(*Daniel Added*)
					myStartLiftDelta := 860 - Move_Height;

					IF Move_Height>(+860)AND Move_Height-860>5 THEN
						Dir:=0;RTSpeed[7]:=16#30;RTSpeed[8]:=16#00;diHomeStep:=1;
					ELSIF Move_Height<(+860)AND 860-Move_Height>5 THEN
						Dir:=1;RTSpeed[7]:=16#30;RTSpeed[8]:=16#00;diHomeStep:=1;
					ELSIF ABS( Move_Height-860)<=5 THEN
						diHomeStep:=7;
					END_IF
					abyRecv:=LanNullArray;
		(*Jog动作*)
				ELSIF(abyRecv[1]=74)AND(abyRecv[2]=79)AND(abyRecv[3]=71)AND(abyRecv[4]=32)AND(abyRecv[5]=76) AND(abyRecv[6]=73)AND(abyRecv[7]=70)AND(abyRecv[8]=84) THEN
					TcpSendData(Client2.diSocket, ADR(str104), LEN(str104), 10);
					TcpSendData(Client2.diSocket, ADR(str105), LEN(str105), 10);
					Temp1:='';
					FOR j:=1 TO SizeOfMsg DO
						Temp1:=CONCAT(Temp1,ASCII_TO_STRING(abyRecv[j]));
					END_FOR
					IF  abyRecv[SizeOfMsg]=16#30 THEN
						Dir:=1;
					ELSIF abyRecv[SizeOfMsg]=16#31 THEN
						Dir:=0;
					END_IF
					IF STRING_TO_UINT (DELETE(DELETE(Temp1,9,(SizeOfMsg-8)),16,1))<100 THEN
						RTSpeed[7]:=STRING_TO_BYTE (DELETE(DELETE(Temp1,9,(SizeOfMsg-8)),16,1));
						RTSpeed[8]:=16#00;
					ELSIF STRING_TO_UINT (DELETE(DELETE(Temp1,9,(SizeOfMsg-8)),16,1))>=100 THEN
						RTSpeed[7]:=16#00;
						RTSpeed[8]:=16#01;
					END_IF
					diJogStep:=1;
					abyRecv:=LanNullArray;
			(*Moveto动作*)
				ELSIF(abyRecv[1]=77)AND(abyRecv[2]=79)AND(abyRecv[3]=86)AND(abyRecv[4]=69)AND(abyRecv[5]=84) AND(abyRecv[6]=79)AND(abyRecv[7]=32)AND(abyRecv[8]=76) AND(abyRecv[9]=73)AND(abyRecv[10]=70)AND(abyRecv[11]=84)THEN
					TcpSendData(Client2.diSocket, ADR(str108), LEN(str108), 10);
					TcpSendData(Client2.diSocket, ADR(str109), LEN(str109), 10);
					Temp1:='';
					FOR j:=1 TO SizeOfMsg DO
						Temp1:=CONCAT(Temp1,ASCII_TO_STRING(abyRecv[j]));
					END_FOR
					FOR k:=19 TO SizeOfMsg DO
						IF abyRecv[k]=16#3B THEN
							SecondColonPos:=k;
						END_IF
					END_FOR
					IF STRING_TO_UINT(DELETE(DELETE(Temp1,SizeOfMsg-SecondColonPos+1,SecondColonPos),19,1))<100 THEN
						RTSpeed[7]:=STRING_TO_BYTE (DELETE(DELETE(Temp1,SizeOfMsg-SecondColonPos+1,SecondColonPos),19,1));
						RTSpeed[8]:=16#00;
					ELSIF STRING_TO_UINT(DELETE(DELETE(Temp1,SizeOfMsg-SecondColonPos+1,SecondColonPos),19,1))>=100 THEN
						RTSpeed[7]:=16#00;
						RTSpeed[8]:=16#01;
					END_IF
					IF STRING_TO_REAL (DELETE(Temp1,(SecondColonPos+9),1))<Move_Height AND Move_Height-STRING_TO_REAL (DELETE(Temp1,(SecondColonPos+9),1))>5 THEN
						Dir:=0;diMovetoStep:=1;
					ELSIF STRING_TO_REAL (DELETE(Temp1,(SecondColonPos+9),1))>Move_Height AND STRING_TO_REAL (DELETE(Temp1,(SecondColonPos+9),1))-Move_Height>5 THEN
						Dir:=1;diMovetoStep:=1;
					ELSIF ABS(STRING_TO_REAL (DELETE(Temp1,(SecondColonPos+9),1))-Move_Height)<=5 THEN
						diMovetoStep:=4;
					END_IF
					TargetPosition:=STRING_TO_REAL (DELETE(Temp1,(SecondColonPos+9),1));(*目标位置（绝对位置）*)

					(*Daniel Added*)
					myStartLiftDelta := TargetPosition - Move_Height;

					abyRecv:=LanNullArray;
				END_IF
			END_IF
		END_IF
	ELSIF diReceived<0 THEN
		CloseSocket(ADR(Client2.diSocket));
		Client2.stIPAddress:= '';
		AutoSendMsgDelay(IN:=FALSE);
	END_IF
	IF AutoSendMsgStep=0 THEN
		AutoSendMsgDelay(IN:=TRUE,PT:=t#500ms);
		IF AutoSendMsgDelay.Q THEN
			AutoSendMsgStep:=1;
			AutoSendMsgDelay(IN:=FALSE);
		END_IF
	END_IF
	IF AutoSendMsgStep=1 THEN
		SendLiftHeight:=CONCAT(CONCAT('GET LIFT;COMPLETED;POSITION=',LREAL_TO_STRING(LREAL_TO_LREALDOTN(Move_Height,3))),'@');
		IF diJogStep<>0 THEN
			SendLiftSpeed:=CONCAT(CONCAT('GET LIFT;COMPLETED;SPEED=',UINT_TO_STRING(LiftSpeed)),'@');
			TcpSendData(Client2.diSocket, ADR(SendLiftSpeed), LEN(SendLiftSpeed), 10);
		END_IF
		TcpSendData(Client2.diSocket, ADR(SendLiftHeight), LEN(SendLiftHeight), 10);
		AutoSendMsgStep:=0;
	END_IF
END_IF

IF HeartBeatCounts>0 THEN
	HeartBeatTimer(IN:=TRUE,PT:=t#2s);
	IF HeartBeatStep=1 THEN
		HeartBeat:=LanNullArray;
		HeartBeatTimer(IN:=FALSE);
		EmergencyStop:=0;
		HeartBeatStep:=0;
	END_IF
	IF HeartBeatTimer.Q THEN
		HeartBeatStep:=0;
		HeartBeatCounts:=0;
		EmergencyStop:=1;
		HeartBeatTimer(IN:=FALSE);
	END_IF
	IF HeartBeatCounts=32767THEN
		HeartBeatCounts:=1;
	END_IF
END_IF
IF EmergencyStop=1AND(diHomestep+ diJogstep+diMovetostep<>0)THEN
	diStopstep:=2;
	diHomestep:=0;
	diJogstep:=0;
	diMovetostep:=0;
	StartCheckSpeed:=FALSE;
	EmergencyStop:=0;
ELSIF EmergencyStop=1AND(diHomestep+ diJogstep+diMovetostep+diStopStep=0)THEN
	EmergencyStop:=0;
END_IF
CASE diHomeStep OF
1:
	FOR m:=1 TO 8 DO
		NeedCRCBytes[m]:=BYTE_TO_WORD(RTSpeed[m]);
	END_FOR
	RTSpeed[9]:=WORD_TO_BYTE(CRC(NeedCRCBytes,8)MOD 256);
	RTSpeed[10]:=WORD_TO_BYTE(CRC(NeedCRCBytes,8)/ 256);
	SysComWrite(ComHandle, ADR(RTSpeed), 10, 0);
	diHomeStep:=2;
2:	IF byRead[1]=16#52 AND  byRead[2]=16#54 THEN
		byMyRead:=byRead;
		byRead:=ComNullArray;
	END_IF
	IF byMyRead[1]=16#52 AND  byMyRead[2]=16#54 AND  byMyRead[3]=16#06 THEN
		diHomeStep:=3;
		byMyRead:=ComNullArray;
	ELSIF byMyRead[1]=16#52 AND  byMyRead[2]=16#54 AND byMyRead[3]<>16#06THEN
		diHomeStep:=100;
	END_IF
3:
	LIFTRE[4]:=UINT_TO_BYTE(Dir+1);
	FOR m:=1 TO 5 DO
		NeedCRCBytes[m]:=BYTE_TO_WORD(LIFTRE[m]);
	END_FOR
	LIFTRE[6]:=WORD_TO_BYTE(CRC(NeedCRCBytes,5)MOD 256);
	LIFTRE[7]:=WORD_TO_BYTE(CRC(NeedCRCBytes,5)/ 256);
	SysComWrite(ComHandle, ADR(LIFTRE), 7, 0);
	diHomeStep:=4;
4:
	IF  byRead[1]=16#52 AND  byRead[2]=16#45 THEN
		byMyRead:=byRead;
		byRead:=ComNullArray;
	 END_IF
	IF   byMyRead[1]=16#52 AND  byMyRead[2]=16#45 AND  byMyRead[3]=16#06 THEN
		diHomeStep:=5;
		byMyRead:=ComNullArray;
	ELSIF byMyRead[1]=16#52 AND  byMyRead[2]=16#45 AND  byMyRead[3]<>16#06 THEN
		diHomeStep:=100;
	END_IF
5:
	IF ABS(Move_Height-860) <4THEN                                                          (* 判断外部编码器，到位后发送RS指令*)
		SysComWrite(ComHandle, ADR(LIFTRS), 6, 0);
		diHomeStep:=6;
	ELSE
		(*Daniel Added*)
		IF myStartLiftDelta > 0 THEN
			IF (860 - Move_Height) < -0.5 THEN
				SysComWrite(ComHandle, ADR(LIFTRS), 6, 0);
				diHomeStep:=6;
			END_IF
		ELSE
			IF (860 - Move_Height) > 0.5 THEN
				SysComWrite(ComHandle, ADR(LIFTRS), 6, 0);
				diHomeStep:=6;
			END_IF
		END_IF
	END_IF
6:
	IF  byRead[1]=16#52 AND  byRead[2]=16#53 THEN
		byMyRead:=byRead;
		byRead:=ComNullArray;
	END_IF
	 IF byMyRead[1]=16#52 AND  byMyRead[2]=16#53 AND  byMyRead[3]=16#06 THEN
		diHomeStep:=7;
		byMyRead:=ComNullArray;
	ELSIF byMyRead[1]=16#52 AND  byMyRead[2]=16#53 AND  byMyRead[3]<>16#06 THEN
		diHomeStep:=100;
	END_IF
7..8:
	LiftUseTimer1(IN:=TRUE,PT:=T#300ms);
	IF LiftUseTimer1.Q THEN
		IF	diHomeStep=7 THEN
			TcpSendData(Client2.diSocket, ADR(str102), LEN(str102), 10);
			diHomeStep:=0;
		ELSIF diHomeStep=8 THEN
			TcpSendData(Client2.diSocket, ADR(str103), LEN(str103), 10);
			diHomeStep:=0;
		END_IF
		LiftUseTimer1(IN:=FALSE);
	END_IF
100:
	SysComWrite(ComHandle, ADR(LIFTRS), 6, 0);
	diHomeStep:=8;
END_CASE
CASE diJogStep OF
1:
	FOR m:=1 TO 8 DO
		NeedCRCBytes[m]:=BYTE_TO_WORD(RTSpeed[m]);
	END_FOR
	RTSpeed[9]:=WORD_TO_BYTE(CRC(NeedCRCBytes,8)MOD 256);
	RTSpeed[10]:=WORD_TO_BYTE(CRC(NeedCRCBytes,8)/ 256);
	SysComWrite(ComHandle, ADR(RTSpeed), 10, 0);
	diJogStep:=2;
2:	IF  byRead[1]=16#52 AND  byRead[2]=16#54 THEN
		byMyRead:=byRead;
		byRead:=ComNullArray;
	END_IF
	IF byMyRead[1]=16#52 AND byMyRead[2]=16#54 AND byMyRead[3]=16#06  THEN
		diJogStep:=3;
		byMyRead:=ComNullArray;
	ELSIF byMyRead[1]=16#52 AND byMyRead[2]=16#54 AND byMyRead[3]<>16#06THEN
		diJogStep:=100;
	END_IF
3:
	LIFTRE[4]:= UINT_TO_BYTE (Dir+1);
	FOR m:=1 TO 5 DO
		NeedCRCBytes[m]:=BYTE_TO_WORD(LIFTRE[m]);
	END_FOR
	LIFTRE[6]:=WORD_TO_BYTE(CRC(NeedCRCBytes,5)MOD 256);
	LIFTRE[7]:=WORD_TO_BYTE(CRC(NeedCRCBytes,5)/ 256);
	SysComWrite(ComHandle, ADR(LIFTRE), 7, 0);
	StartCheckSpeed:=TRUE;(*开启速度检测*)
	diJogStep:=4;
4:	IF  byRead[1]=16#52 AND  byRead[2]=16#45 THEN
		byMyRead:=byRead;
		byRead:=ComNullArray;
	END_IF
	IF byMyRead[1]=16#52 AND byMyRead[2]=16#45 AND byMyRead[3]=16#06 THEN
		diJogStep:=5;
		byMyRead:=ComNullArray;
	ELSIF byMyRead[1]=16#52 AND byMyRead[2]=16#45 AND byMyRead[3]<>16#06 THEN
		diJogStep:=100;
	END_IF
5:	IF (ABS(RTSpeed[7]+100*RTSpeed[8]-LiftSpeed))<5 THEN
		LiftUseTimer1(IN:=TRUE,PT:=T#300ms);
		IF LiftUseTimer1.Q THEN
			diJogStep:=6;
			StartCheckSpeed:=FALSE;
			TcpSendData(Client2.diSocket, ADR(str106), LEN(str106), 10);
			LiftUseTimer1(IN:=FALSE);
		END_IF
	END_IF
7..8:
	SysComWrite(ComHandle, ADR(LIFTRS), 6, 0);
	IF diJogStep=7 THEN
		diJogStep:=9;
	ELSIF  diJogStep=8 THEN
		diJogStep:=10;
	END_IF
9..10:
	IF  byRead[1]=16#52 AND  byRead[2]=16#53 THEN
		byMyRead:=byRead;
		byRead:=ComNullArray;
	END_IF
	IF  byMyRead[1]=16#52 AND byMyRead[2]=16#53 AND  byMyRead[3]=16#06 THEN
		SendTimes:=0;
		LiftUseTimer2(IN:=FALSE);
		byMyRead:=ComNullArray;
		IF diJogStep=9 THEN
			diJogStep:=11;
		ELSIF  diJogStep=10 THEN
			diJogStep:=12;
		END_IF
	ELSIF  byMyRead[1]=16#52 AND byMyRead[2]=16#53 AND byMyRead[3]<>16#06THEN
		diJogStep:=100;
	END_IF
11..12:
	IF diJogStep=11 THEN
		TcpSendData(Client2.diSocket, ADR(str127), LEN(str127), 10);
		diJogStep:=0;
	ELSIF diJogStep=12 THEN
		TcpSendData(Client2.diSocket, ADR(str128), LEN(str128), 10);
		diJogStep:=0;
	END_IF
13:
	LiftUseTimer1(IN:=TRUE,PT:=T#300ms);
	IF LiftUseTimer1.Q THEN
		TcpSendData(Client2.diSocket, ADR(str107), LEN(str107), 10);
		diJogStep:=0;
		StartCheckSpeed:=FALSE;
		LiftUseTimer1(IN:=FALSE);
	END_IF
100:
	SysComWrite(ComHandle, ADR(LIFTRS), 6, 0);
	diJogStep:=13;
END_CASE
IF diJogStep>0 AND diJogStep<=6  THEN
	Vert_Limit_Up:=1-(DINT_TO_WORD(Input_Value) AND 64)/64;			(*升降：上限位开关*)
	Vert_Limit_Down:=1-(DINT_TO_WORD(Input_Value) AND 128)/128;	(*升降：下限位开关*)
	IF Vert_Limit_Up=1 AND Dir=1 THEN
		diJogStep:=7;
	ELSIF Vert_Limit_Down=1 AND Dir=0 THEN
		diJogStep:=8;
	END_IF
END_IF
(*MOVETO LIFT*)
CASE diMovetoStep OF
1:
	FOR m:=1 TO 8 DO
		NeedCRCBytes[m]:=BYTE_TO_WORD(RTSpeed[m]);
	END_FOR
	RTSpeed[9]:=WORD_TO_BYTE(CRC(NeedCRCBytes,8)MOD 256);
	RTSpeed[10]:=WORD_TO_BYTE(CRC(NeedCRCBytes,8)/ 256);
	SysComWrite(ComHandle, ADR(RTSpeed), 10, 0);
	diMovetoStep:=2;
2:	IF  byRead[1]=16#52 AND  byRead[2]=16#54 THEN
		byMyRead:=byRead;
		byRead:=ComNullArray;
	END_IF
	IF byMyRead[1]=16#52 AND byMyRead[2]=16#54 AND byMyRead[3]=16#06  THEN
		diMovetoStep:=3;
		byMyRead:=ComNullArray;
	ELSIF byMyRead[1]=16#52 AND byMyRead[2]=16#54 AND byMyRead[3]<>16#06THEN
		diMovetoStep:=100;
	END_IF
3:	LIFTRE[4]:= UINT_TO_BYTE (Dir+1);
	FOR m:=1 TO 5 DO
		NeedCRCBytes[m]:=BYTE_TO_WORD(LIFTRE[m]);
	END_FOR
	LIFTRE[6]:=WORD_TO_BYTE(CRC(NeedCRCBytes,5)MOD 256);
	LIFTRE[7]:=WORD_TO_BYTE(CRC(NeedCRCBytes,5)/ 256);
	SysComWrite(ComHandle, ADR(LIFTRE), 7, 0);
	diMovetoStep:=4;
4:	IF  byRead[1]=16#52 AND  byRead[2]=16#45 THEN
		byMyRead:=byRead;
		byRead:=ComNullArray;
	END_IF
	IF byMyRead[1]=16#52 AND byMyRead[2]=16#45 AND byMyRead[3]=16#06 THEN
		diMovetoStep:=5;
		byMyRead:=ComNullArray;
	ELSIF byMyRead[1]=16#52 AND byMyRead[2]=16#45 AND byMyRead[3]<>16#06 THEN
		diMovetoStep:=100;
	END_IF
5:	IF ABS(TargetPosition-Move_Height)<5 THEN
		diMovetoStep:=6;
	ELSE
		(*Daniel Added*)
		IF myStartLiftDelta > 0 THEN
			IF (TargetPosition - Move_Height ) < -0.5 THEN
				SysComWrite(ComHandle, ADR(LIFTRS), 6, 0);
				diMovetoStep:=6;
			END_IF
		ELSE
			IF (TargetPosition - Move_Height ) > 0.5 THEN
				SysComWrite(ComHandle, ADR(LIFTRS), 6, 0);
				diMovetoStep:=6;
			END_IF
		END_IF
	END_IF
6:
	SysComWrite(ComHandle, ADR(LIFTRS), 6, 0);
	diMovetoStep:=7;
7:	IF byRead[1]=16#52 AND  byRead[2]=16#53 THEN
		byMyRead:=byRead;
		byRead:=ComNullArray;
	END_IF
	IF byMyRead[1]=16#52 AND  byMyRead[2]=16#53 AND  byMyRead[3]=16#06  THEN
		diMovetoStep:=8;
		byMyRead:=ComNullArray;
	ELSIF byMyRead[1]=16#52 AND  byMyRead[2]=16#53 AND  byMyRead[3]<>16#06 THEN
		diMovetoStep:=100;
	END_IF
8..9:
	LiftUseTimer1(IN:=TRUE,PT:=T#300ms);
	IF LiftUseTimer1.Q THEN
		IF	diMovetoStep=8 THEN
			TcpSendData(Client2.diSocket, ADR(str110), LEN(str110), 10);
			diMovetoStep:=0;
		ELSIF diMovetoStep=9 THEN
			TcpSendData(Client2.diSocket, ADR(str111), LEN(str111), 10);
			diMovetoStep:=0;
		END_IF
		LiftUseTimer1(IN:=FALSE);
	END_IF
100:
	SysComWrite(ComHandle, ADR(LIFTRS), 6, 0);
	diMovetoStep:=9;
END_CASE
(*STOP LIFT RS232通讯*)
CASE diStopStep OF
1:	LiftUseTimer1(IN:=TRUE,PT:=T#300ms);
	IF LiftUseTimer1.Q THEN
		TcpSendData(Client2.diSocket, ADR(str113), LEN(str113), 10);
		diStopStep:=2;
		LiftUseTimer1(IN:=FALSE);
	END_IF
2:
	SysComWrite(ComHandle, ADR(LIFTRS), 6, 0);
	diStopStep:=3;
3:	IF  byRead[1]=16#52 AND  byRead[2]=16#53 THEN
		byMyRead:=byRead;
		byRead:=ComNullArray;
	END_IF
	IF  byMyRead[1]=16#52 AND byMyRead[2]=16#53 AND  byMyRead[3]=16#06 THEN
		diStopStep:=4;
		byMyRead:=ComNullArray;
	ELSIF  byMyRead[1]=16#52 AND byMyRead[2]=16#53 AND byMyRead[3]=16#06 THEN
		diStopStep:=100;
	END_IF
4..5:
	LiftUseTimer1(IN:=TRUE,PT:=T#300ms);
	IF LiftUseTimer1.Q THEN
		IF diStopStep=4 THEN
			TcpSendData(Client2.diSocket, ADR(str114), LEN(str114), 10);
			diStopStep:=0;
		ELSIF	diStopStep=5 THEN
			TcpSendData(Client2.diSocket, ADR(str116), LEN(str116), 10);
			diStopStep:=0;
		END_IF
		LiftUseTimer1(IN:=FALSE);
	END_IF
100:
	SysComWrite(ComHandle, ADR(LIFTRS), 6, 0);
	diStopStep:=5;
END_CASE
CheckLiftSpeed(Execute:=StartCheckSpeed, recieve:=byread,RG:=RG,SPEED=>LiftSpeed);(*推杆实时速度*)
END_PROGRAM

(* POU 子程序/SensorRead, ST *)
PROGRAM SensorRead
VAR
	Lift_ADC,Tilt_ADC:INT;
	Lift_AVG,Tilt_AVG:DWORD;
	i,j:INT;
	myAvgSampleCount:INT:=5;
	Lift_Angle: REAL;

END_VAR
IF j< myAvgSampleCount THEN
	GT_GetAdcValue(1, ADR(Lift_ADC), 1, 0);
	Lift_AVG:=Lift_AVG+Lift_ADC;
	j:=j+1;
ELSE
	Lift_AVG:=Lift_AVG/myAvgSampleCount;
	(*Lift_Angle:=(Lift_AVG-13107.2)/145.635;*)
	Lift_Angle:=(Lift_AVG * 225.0 ) / 65536;

	(*If the lift is moving, update real angle. If the lift is stoppped, then do noise band check*)
	IF gLiftMotionState = 0 THEN
		IF ABS(gLastLiftAngle - Lift_Angle) < 0.4 THEN
			Lift_Angle := gLastLiftAngle;
		ELSE
			gLastLiftAngle := Lift_Angle;
		END_IF
	END_IF

	Move_Height:=800*SIN(ABS(Lift_Angle)*0.0175)+275;
	Lift_AVG:=0;
	j:=0;
END_IF

IF i<myAvgSampleCount THEN
	GT_GetAdcValue(2, ADR(Tilt_ADC), 1, 0);
	Tilt_AVG:=Tilt_AVG+Tilt_ADC;
	i:=i+1;
ELSE
	Tilt_AVG:=Tilt_AVG/myAvgSampleCount;
	Move_Angle:=(Tilt_AVG-13107.2)/436.907;
	(*Move_Angle:=(Tilt_AVG*225.0)/65536-45.0;*)
	Tilt_AVG:=0;
	i:=0;
END_IF
END_PROGRAM

(* POU PLCOpen_CAN2.3/运动控制功能块/SDORead, ST *)
FUNCTION_BLOCK SDORead
VAR_INPUT
	xEnable			: BOOL;				(*Rising edge enable the FB to send one SDO*)
	byNodeID		: BYTE;				(*Station ID*)
	wIndex			: WORD;			(*index to write data*)
	bySubIndex	: BYTE;				(*subindex to write data*)
	tTimeOut		:TIME:=t#100ms;	(*after this time, if there was no answer, there will be an error code*)
END_VAR
VAR_OUTPUT
	xDone			: BOOL;			(*SDO answer received*)
	dwData			: DWORD;			(*Read Data*)
	xError			: BOOL;			(*error happend*)
	iErrCode			: INT;			(*0:normal	1:timeout	2:date length error*)
END_VAR
VAR
	RTrig:R_TRIG;
	FTrig:F_TRIG;
	SDO:CanOpenSendSDO;	(*SDO-mode, use 16#40 FOR read-request,
		use 16#23 FOR 4-BYTE-write-request.
		use 16#27 for 3-byte...
		use 16#2B for 2-byte...
		use 16#2F for 1-byte...
		use 16#21 FOR downloading more than 4 bytes using the segmented transfer.*)
	iStep: INT := -1;
	byModus: BYTE := 00;
	Timer: TON;
END_VAR
RTrig(CLK:=xEnable);
FTrig(CLK:=xEnable);

IF RTrig.Q THEN
	xDone:=FALSE;
	xError:=FALSE;
	iErrCode:=0;
	byModus:=16#40;
	iStep:=0;
END_IF

IF FTrig.Q THEN
	SDO(Enable:=FALSE);
	iStep:=-1;
END_IF

CASE iStep OF
0:
	SDO(
		Enable:=TRUE ,
		wDrvNr:=0 ,
		ucNodeId:=byNodeID ,
		wIndex:=wIndex ,
		bySubIndex:=bySubIndex ,
		ucModus:=byModus ,
		aAbortCode:= ,
		dwDataBufferLength:= ,
		pDataBuffer:= , 
		bWaitForAnswer=> ,
		bAnswerRec=> , 
		ucAnswerBytes=> , 
		iAnswerLength=> , 
		bToggleUnequal=> ,
		bAbortRec=> ,
		aAbortRec=> ,
		dwReadDataLen=> );
	iStep:=1;
1:
	SDO();
	Timer(IN:=TRUE, PT:=tTimeOut);
	IF SDO.bAnswerRec THEN
		iStep:=-1;
		xDone:=TRUE;
		dwData:=BYTE_TO_DWORD(SDO.ucAnswerBytes[4]) OR SHL(BYTE_TO_DWORD(SDO.ucAnswerBytes[5]), 8)
			OR SHL(BYTE_TO_DWORD(SDO.ucAnswerBytes[6]), 16) OR SHL(BYTE_TO_DWORD(SDO.ucAnswerBytes[7]), 24);
		SDO(Enable:=FALSE);
		Timer(IN:=FALSE);
		RETURN;
	END_IF
	IF Timer.Q THEN
		iStep:=-1;
		iErrCode:=1;
		xError:=TRUE;
		SDO(Enable:=FALSE);
		Timer(IN:=FALSE);
	END_IF
END_CASE
END_FUNCTION_BLOCK

